(* CoDeSys 2.3 project: cy-wg-016-001.pro *)
(* Title: cy-wg-06 - ClevergyAS *)
(* Author: Andrea Ravasio *)
(* Libraries: Standard.lib 2.12.10 13:48:34, Util.lib 26.9.14 09:12:46, Visual.lib 2.12.10 13:48:34, WagoLibIdent.lib 25.2.13 10:12:16, WagoLibStatus.lib 2.12.10 13:48:32, SysLibFile.lib 2.12.10 13:48:34, SysLibRtc.lib 2.12.10 13:48:32, SysLibSockets.lib 10.2.11 08:20:54, SysLibEvent.lib 2.12.10 13:48:34, SysLibPlcCtrl.lib 2.12.10 13:48:32, SysLibCallback.lib 2.12.10 13:48:32, mod_com.lib 2.12.10 13:48:32, SerComm.lib 31.5.11 07:54:36, Serial_Interface_01.lib 22.4.13 11:50:14, Modb_l05.lib 22.4.13 11:50:12, Ethernet.lib 2.12.10 13:48:32, MBus_03.lib 9.2.13 16:51:58, WagoLibModbus_IP_01.lib 26.5.15 10:20:08, WagoLibMBX_01.lib 20.3.12 15:32:40, LON_01.lib 28.9.12 13:05:10 *)

(* PLC configuration (modules and I/O channels)
VPN_ST2 AT %IX36.0 [BOOLOnX_I] Ch_1 Digital input
LAMP_AL AT %QX22.0 [BOOLOnX_Q] Ch_1 Digital output
KEY_QE_ST AT %IX36.1 [BOOLOnX_I] Ch_2 Digital input
CIR01_EN AT %QX22.1 [BOOLOnX_Q] Ch_2 Digital output
CIR05_AL AT %IX36.2 [BOOLOnX_I] Ch_3 Digital input
AT %QX22.2 [BOOLOnX_Q] Ch_3 Digital output
CIR05_AUTO AT %IX36.3 [BOOLOnX_I] Ch_4 Digital input
AT %QX22.3 [BOOLOnX_Q] Ch_4 Digital output
CIRD02_B_AL AT %IX36.4 [BOOLOnX_I] Ch_5 Digital input
AT %QX22.4 [BOOLOnX_Q] Ch_5 Digital output
CIRD02_B_AUTO AT %IX36.5 [BOOLOnX_I] Ch_6 Digital input
AT %QX22.5 [BOOLOnX_Q] Ch_6 Digital output
CIRD02_A_AL AT %IX36.6 [BOOLOnX_I] Ch_7 Digital input
AT %QX22.6 [BOOLOnX_Q] Ch_7 Digital output
CIRD02_A_AUTO AT %IX36.7 [BOOLOnX_I] Ch_8 Digital input
AT %QX22.7 [BOOLOnX_Q] Ch_8 Digital output
0750-9999/0400-0008 8 DI Generic [Type_1_8_Channels] node 1, in %IB72 out %QB44 {INTTypePAAssignment = PLC; INTTypeModule = plugged}
  CIRD01_B_AL AT %IX36.8 [BOOLOnX_I] I 1: Digital Input
  CIR01_AL AT %IX36.9 [BOOLOnX_I] I 2: Digital Input
  CIRD01_B_AUTO AT %IX36.10 [BOOLOnX_I] I 3: Digital Input
  CIR01_ST AT %IX36.11 [BOOLOnX_I] I 4: Digital Input
  CIRD01_A_AL AT %IX36.12 [BOOLOnX_I] I 5: Digital Input
  CIR01_AUTO AT %IX36.13 [BOOLOnX_I] I 6: Digital Input
  CIRD01_A_AUTO AT %IX36.14 [BOOLOnX_I] I 7: Digital Input
  CIR04_AL AT %IX36.15 [BOOLOnX_I] I 8: Digital Input
  CIR04_AUTO AT %IX37.0 [BOOLOnX_I] I 1: Digital Input
  CIR02_AUTO AT %IX37.1 [BOOLOnX_I] I 2: Digital Input
  CIR03_AL AT %IX37.2 [BOOLOnX_I] I 3: Digital Input
  CTL01_ST AT %IX37.3 [BOOLOnX_I] I 4: Digital Input
  CIR03_AUTO AT %IX37.4 [BOOLOnX_I] I 5: Digital Input
  CTL02_ST AT %IX37.5 [BOOLOnX_I] I 6: Digital Input
  CIR02_AL AT %IX37.6 [BOOLOnX_I] I 7: Digital Input
  AT %IX37.7 [BOOLOnX_I] I 8: Digital Input
0753-0648 LON-FTT [Type_55_1_Channels] node 3, in %IB0 out %QB0 {INTTypePAAssignment = PLC; INTTypeModule = plugged; DataStream = 1F8B0800000000000400ED7D7B6FE2C8D2F7FF8FF47E073F48CFD18C14261808B99C242B0F98095AC0395C921DCD8C90631AF08EB139BE2493FDF46F75B76D6CDCBE10601288A5D52CB1DBD555DDD5BFBA74B97DF9C7AFB9C63D22D3520DFDAAC07F2A1538A42BC658D5A75705C79E14F95AE18FEBFFF73F976D436FE93632; DataStream = 27B282387848B72E7E59EA556166DB8B8BE3E3A7A7A74F4F954F86393D2E974AFCF15F9D765F99A1B95C5475CB96750515FCA7C6E94F15B85BD3989AF2BC058DCF4B17A5D2C529FC7B7251E22F4AB58B52157E14B8BFD449579EA3ABC2BD3C354677AA6DD8A6A1AB4AA50462F4913669188A3347BA2DDB205EDD98E3DF5705; DataStream = 613CE69E0DC7E4147A859B2113D8EB22079E6EAAE6FC4936D19D3F26E7A4A3BEFC886E657B7655A85F7CFFA2DADF95E76289AF159FA6DC8706B290FE8FAC1BDCADACC9FFFC63701D07D85017B28638A1C40B1FBFB7A5EE48474F05AE638C1D0D759DF90332817801C696E3F0E87664F3A7F4F037526C8B5C5BBDEA5E84CB03; DataStream = 345F68B28D5A63605E9DA8C8F4EFC15D3C70ADF175A9C4B1FEBB3C76EF079EE82BC6025DC32DFA2370E74FF48CAFE3FF05AEB6F431FA75CD5F1ED31F3E5FC7098CF94CE309BBEE376F07BA314654B2E583E4A6FF08B369B88964AA5355973566D3D04DFF9196D536949F687C6D9B0E0219BC3F030D3AB23E966DC37CF6DB2C; DataStream = AF049A490BAC56B2763D91358B34F3AFF8AD3A084F349D6E3C94A1BFFD56A286B022D60D07B41196D585AE6A5705DC79813B0E0C08B29F0CF3E79D6CAAF28386ACE0A4ACDC0BDC4AD39897694DB2E6F8DA735E5E559F800AE19B611D4AD523862E75EF0623E3E1EF9189FEEB202B4E9B961AA53FAA3DAF69B4494869824D99; DataStream = DA9449A3D6D0AAEC9A15D52E3E46BB48CB6C1A4689AA7A1FE9E3813A27531BFC33DC4EFE156A17F873B55D0F29487D4481A6C12B2BC2DF9AAA61AAF6F35278FF4AA8651F998FAA8206CFA07982F253379E34349EA2316863E04EE891866A0232C0405EB7F4850393BABC1066190CE04455F0DC5C770D1D98085E0935AD1BFA; DataStream = 449D3A263131B04A16C8B45564AD0E6ACBF2BB5A5196D5EBA1C73E3FDBA8AFFE83AE2B97C7FEEFC0AA3F8E5FF66F16112A498850D9262280E3613B56064030FA6ECB543CF05BBE793828E770901D0E24C7DE2F3CA81D0C1E9C26E1C1E9D6F060A26A08BB0859DC8326B4EDE1A6E9EE81DF748B78E02B7A3A20782433E0C149; DataStream = 8E0787EB1EF0E5C3C1836A121E54B78A07D91D04BCCEB1E9CFE2222CDBBE7950A8E5A070C04E42F9F46050E13C9286A22344A386D25651616164810462FA6F8D2C41C3B2E99B0784D31C100ED74B58376888DC59661C5359BE3C6665AF5F96D24E4E5017F9980C7571CD1435599477AA693BB2C64D1C5DA1AB857BD0605057; DataStream = 33CF6BA59113D66A9E47CE86FF6F2F8F0CCDB3E691A3B43318025F1BB66809D64920C5691969999B02EEADF986BE787946998ED0EB6594A175C68C7284720E0C87050CAFEF23AE890B8793593E4BCA249D6D2D9364836AE1E53B5F64C105AC887D94D1650892CE81E1B08061FF3C86C3C9269D9D2521C3D9B69041D664739E; DataStream = 051404DA300B24B8347334382C34D83B37A17C9EA3C12ED120B38F9003C24102C2FEB907878408491985B3AD651470CC8F32E519B5E73E6D9B05115CB239221C1622EC9F8B703078C097925C0472773B88307B9495D1DC186742859B7A9D1FC12C67CF2704C8E7E87058E8B07FFE029FC3C3EF81871C1BDE3936EC9DE77048; DataStream = D07092080D275BDB85802BA34C3B10041770B3ECDB102EED1C170E0B17F6CF6738A490E2ED02438E0AEF1915F6CE5BC84161D7A0D077168B1C18DE3B30E4EE429E62700769090EE53C0399C3C39EC2C321A519DE343CE4D8F0CEB161EF628A438286B7185394F30C648E0BFBE8331C5248F17681214785F78C0A7BE72DE4A0; DataStream = B06B50C833903930E4EE429E62F00769090E953C0399C3C39EC2C321A519DE343CE4D8F0CEB161EF628A438286B7185354F20C648E0BFBE8331C5248F17681214785F78C0A7BE72DE4A0B06B50C833903930E4EE429E62F007C90587C6CD7D9E80CCD1614FD121CF32ECD06FC0D0202876EE35BC775CC8C3891C16C2B000DE; DataStream = C2ADA1EA79F2F15DE3C2FEF90B3930EC1818F24D891C17727FE1F560E13C0915CEB7060AD6936A2BB32CA0506F36B0B720EA7894321E00E912CF61E1B060217717725C08E1C2971C17725CC8DD857C4FC21BA4B0CF90173EE6E0B0874E43BE27B1C31C0386867C43E2BD8342EE31E498107117F20D89778F0BFBE72CE4C0B0; DataStream = 7B60C8FD85F78E0BB9BF90271E3D50F82CD5F30D891C16727781CB71815BC1857C4322C785DC5DC83724FC410AFB0CF986440E0E7BE834E41B123BCC316068C8130CEF1D14728F21C78488BB906F48BC7B5CD83F67210786DD0343EE2FBC775C38787F2172C75ADE4AE3F9F2B86DE81DD9FC293DFC0DAC91AB2BD7ACEBCBFF; DataStream = FD566F0803E1DBE51FBFE61AF7884C0BA85D15F84FA502877405064C9F5E151C7B52E46B853FAE2FEBB22D6BC6F4FAB2A96A886B59F03F1B99680C8F14B806DCBCF34954310DDC0C4FE15501FF0B7F1BE65CB6FD4635DCA623FF6D9881E70ADCAD6CCFAE0AF58BEF18B54C794EC858DC875F67B58FDF41847B1812EB3BA668; DataStream = 7DEF0F846E43E8353E0DBEDEC29304E6AE0A313858E07A6802FCEA0A4A6C8555BA6FCBF305F0533EE62BC7E5125FE6F8B38B72E9822F17AE57D19AB0C2BCCA7D962D7704FAB05215FB5BED4781234B18C42F70043CAF0AA795028761E9AA4006D644FF759065C3B5479B3E8C710C241447FD416F581F50496168603455853E; DataStream = 49B06E028F8FE0F10287B50CB35FE086BA0A9DFD4BB3FFDDD21F654D1D73966DC2C4423796E1980AFAD7D4FE375BA800FBA2EECC398F3CE66E64E3B9FBA5CE9D3911054086FE2EF29E30BD7839C4EEB0C392C217BDAF4E7557B15C513C49268121E27478CA2A70983B4417833BA427181453641AEA16E905746A0A7361B574; DataStream = 1B4D9149FA6A597D45D664FAC752CE9393CA89271EE98925DCB0DB6F7DE98A8D515BEA7E2970D26462219B108A0AAC5222B8332404C42D87C4755BED5A2217D2391B1680E130272E46B60A7B3209B9914F2E5ECAB9AA69AA8514431F5B99E48499FE5659AE257F0135402BC0CA634DE0E4F11874DC628BD192BA4BF64F58EC; DataStream = 8FB196FB3428C3271EC31E0EF99D645CFFE525CF658F678192E06CFC1800AF6D3E27ADFD44A6313BB6C76DC5E396D543565DEACF0C4C318B32552A011CA85422F2112390A053FD1BA99726202512D1241F1ECE8A0FAACD392EF31C201E759076BB72C203ACAE890CB51721035F8B1375D571206ED44BEC936B5A9C071DD945; DataStream = DD18A3A43595493F2D3D7E29598C7E76A0A57C4049F97DD2D1CFAAED4FCE8A402EF8197359D559EC7F6E0D9A29FA36761F8E67DB9F28DA746DABC49D724404F82760135D814E8302954F3D91BAA00C2F1448278FC68B43F44C2791D63A42542342547D21AA4121026615F09653709374514ED99694D884045988189C31E170; DataStream = 53156533A22F966860CABA25939087380B66BA5C67CC85F26BE43E1E2F1A6900A30793B52E98AF010AE5939330DCAD0302E74CA473C9C44B465B04557003E03EFD115C4A94852FA6E12C3686ECE9221EB2A7A11E3606B034140EABD48BB0F7C1303424EBBB80ADDA5285A0CF17F26F91473380301D7ADAFCDD9B0ECAC75077; DataStream = 2C683B5191367EA1280E2191244A5A249D9B92DC94840078634B32A554365349B6697989C17999CBED02BC63CFF09E804223748389387183C39798112F901C1989E8B33EE6BF44362FC7BDAE54CCBCD00288AD21D5068E43F54770857A19C96A282369D9B2ED247A10490949EF69377E3DDD7E4E92F6104A49F23C3327D98F; DataStream = 95242E25B9E43E3123499BC527246BBB4F42747DE4C61CC5E4BDB2A726A921181993914B2E3E15E11AA45D0BD8471A526C62E1B5E4283D4376D272898D28B1AD656071663221CBF7D26CA43C367DCEB696D57721202691AA98EAC23698063953E0300E90D836E78269CACFDFF8DA0FACEE4D3A43138393F1650ED1ADD2A5C7; DataStream = 8BB75A2CF24800AFFDA758020ABD9EF035453E023D94808B08354F3CCA07B0C6D73865269BE0E02033439298AC8E3A3C90D1F660300DA05CF92C22DCEA9030E6922E99FA8DD05B0A5C66DA5A5FE26FFCC98F953513878E34D925F4EBADD672285E6EB4483FFF71E47146678CAF9E56CF2AB5EA695A6CE60EC37F864223300C; DataStream = 4C6464C4682BD2577D23FD6CAFE541BF1019076969CB302096D7099D33AFD9AD3A22A9A099793B24B07D73BE5DF8A1E8434367AED588411F26F8F80FBD147C68203D52C79E6C51ECA97154FB761BE3C48ABFA963EF4BF82D8235D9B2E9BF29B8A9AD8C8486F4A93DDB3C0470E5F7C8C50F80D8E5F8EA79E9ACC87BE915EF99; DataStream = 379729C50509DB49956E3F8E4BDF7488958AE960AEBBFFB04E84BE01CCF2812D3E7E59837256098648887B04E738D9F78B09F9702084189B95D885561FD5B1236B1C5EB0649D6E21674CD9C5144BF1A9A328AFF040693B3983F8C4640ABFFC9AFCF2BBE1B79C95DFF29AFC9677C36F252BBF9535F9ADEC86DF6A567EAB6BF2; DataStream = 5BDD0DBF2759F93D5993DF93DDF05BCBCA6F6D4D7E6BBBE1F7342BBFA76BF27BBA457EB37178969EAC67BA36F0ECD92B83EFF9CB593F7F651CE6130C5D1AEFFC8E8C5E6650E613AC5E2AF33BB28099119A4F3081A9CCEFC81C66866B3EC11EA632BF23DB9819BBF904E398CAFC8E0C656620E7132C652AF399ADE6D6AAFEBC; DataStream = 88C0CFC2E08278BCC13167EE65A6C40378D375E43E4CB9F737809E916C1E717343B76747DC587E3EE2668683AFA8BA63A3238E160467CC9A66CF9C554AB8CA9FB139F415C9EC882798438B8AF94C1E4B4A07968312AF930E5C2B7EF5C4E8E0015D277E6506E5734A255EF748831D09535926CA646631749C28CC487C2C2756; DataStream = 3CC0ED1D8951F683EA1B50EC75E4A8B2E4981122F182E0FB3B92E4E4DCD72EB23837AE919DBB6412F48BB4D8B93C7D0A326BC8C32C1C72B12A29871578BD6193FC4D204FCE2F77ECCFFCAD1F01849DBF7CCB1E8FD5DC07AE9D64CCDB865BFFB146C2DC7B26215F1E1548F31F7ADD1C799CC01BAE214FBCF512E458E08DF3E3; DataStream = 2FDCA7A2AF1EC66C7BACF376844108D1ED8FD80D2BDA28F3DE3DA92721EA3FC25B61A172924A39E43154C28BCD8ED97EA3352589756BCBFE92365165BF9BF80A93D3AC222EDC42A591861E9196A56AC62F6D224FA44BCA2C630B779B24ED22D45DBCC467BFE9253F0C14DDBB75EA69981B5A440F47B631C2389BA4B7EAB253; DataStream = 4E911D0B83AD0BCBA9F2529CAD129CBDC329F61890ADB240F68EEE9DA5EE48B2B771DC9DB7951D701F6AABBF056A9932AFB195C3045A221929934908C57E2FACD22026396E89D34E26A232A2983D085D7826A8EE67ECC23361730F831776F1D09E462FEC12A03D0E5FCAEC3DF8B5E2976DA3D9F9796086FC57C1D7A9686206; DataStream = FEF320ADADBD7D1E34B1D4FFD3D43978D86B18DAC06319CC2DBB5C8B7A8E2E8DD735BA09A3B0865E26F8C784F466067883903B5CCEEB3A9FE7BEF925B5960BC352E3E2D32C45F2F07C244A5DE0D3CF9079E4D5F3ECBE38B287E4F1F13DF8DE5820D2796AA924E315A3A7D1C24EC988FA9A4AAAABF1D42DDF53DCFD3117BE90; DataStream = 196AB5C238C3CCCB81C0B1555A3EC82CDFAB5AD6846E5D277D47CA0DB45F7E940CC4CEA3C0692CA1E3245A8D239FF21B4A18FCC62C814B9875164EB9CA0CA1D327241C42338D74B8DBA410DA0875171F42E3487543450C6C1E9597BB47E79515C95F9C90C49A187E85A8165444F7C59B89264FB39BB983D1C6D4620D37675B; DataStream = 6C35C810A56F4432154FA554D8BC6F612B95CF2684A7CE5B9064B9867E7F294743B53091F126728C5D1AAF52CE213976D198148957666D2285E1D8F805334AE8558A3BA405D28B8A6A2A8EBA915E194067E4D27995420F774E2C7A72E21626C5A5F42A851F1DA4CC645D858E8B13D9D1369A99B94F6B4468BD4A314813A1F1; DataStream = 83ACFC047154CD31379A9F894B6BE4D2FA4D657FD223328BA6AC4FB332CF0CC90DA03222545EC5920CC1AE6E410A0793D9A518291644C4EFAE9A6BAF0FA62CC8A7B5CBF591625186E49B4145DB28CE916C655F2031B38389E19D1697D8AB5896BA319F3BBA7BD481B5E6C267CAA500C51D2CFAEC36A6097DA331D8186D52B4; DataStream = B33B624C61B01C234C6964EFCC0F4B2B2FF4E428AA7A718139C4870F6D20932FCE48D5471EC157B137F424E22298F24DE4D1089511FBF0CE5DD8988EAC3B80698AA1DBA6A165649D999399134A2397D22B452D0BF0C9E8D6FD0692802A793539BFDFD05019B0D136D57156F08A13C323F32A16A68716866917E7B2F5731331; DataStream = 4C426684C9BC8A55F13852F569117F1D6B1359164B5AE44B5BAF62538202619BB02D8130AD57B12A6433A4A81BB63A792E8ED70BF59952D12D104A70B4DBB83FC5AAF490C57EDF37D3C2817B80C7F3858692774E5F7044DF1917342D7E2924EED37C44E30CAF6D30B7D802CFEFE2F4AD0D12FDCB77B0C907345F9056B5DC07; DataStream = 57F28FA4D4856655D14E760D97652BB1D546AB3B84F1A546EEA478EF487CA619F79509FA3F722492A3695EF95AAA5EF5373953387CD854D25923ABF51F71C74FA51C36E20B4ADA92F3ED363C5FC54D8F7B5B0427190B5FCAA7B5D07934E5D30AEF6F2DE22FB6E0BD0712BBACFD8E45E0532EE1C1F0A6BD9CF4DAC51881278E; DataStream = 2CAE8E344B75B26C31925D1EF2094A3B301067214566CEF9CD9D50E7E6310708C49D3116FEE065D214FBE413B674AAB1B36F5D5F06DA87FFE2965F4E18C853F7AC9FE506D7F525ADAC0B25E439770947256AF646DD61BBC0F5E427D2860ED171984A1F53D76D55D638595170EC6522BC77CD2427DD8ADDD1401AF5C56E2303; DataStream = A527BCBF9B42AA27D6C5D69D18E432CA645D332CC4C93A80BBFC88DCA3C79864EB6DA92F8E9AAD7688623981E218615B984EB321B6C54194742542BA478EEC0436C7E4933486F9EC7D4F8049BDD182211848BDAFB0EEA43F87B741E2D5287160D998AF3955A39E10A47A9242758D695BA14C0FD83B0E683453BD6B41F5F6CF; DataStream = 0D5C57BBFB19B49B9485D8F878D3093239CB210282198A21F857530411FF8C9069F833A919C64F7CE46F1A253A97845692628BA669981C3E85738174ECB5C4AA619F0E7D5368B59335DB27395E613A9953B1D74B56EBF050AA3AB7CCADC48FE5B0DB107BF7B88E2A49A97D96B13EC3281C630D4C198D96B4CA7254ADC32CE3; DataStream = 9720C71CC9A330290E5A1D511A0E56C9D62264EF55582D4F9C45F04E411CC2ECC710BD6F751BD2FD2ACDD308CD954359FD042393A8301CDCAC923C8B92A4AB991A2AC3069D5DE0B019B11103A8D6EB62BF0F5326DCAD28D9790A603CA0670390549498A72200E9BE28FE396A75EF8436DEB60F2C885274CEDCD6F7428BE975; DataStream = 86EF0748F1D9B0E7D4C59ED03B266116868B31F6E1FCF99D815622E6040BEDD18D28808A876128BA7856494E0CC38E25D994A4C12AC9E83A6FA007674A8E17C41FF4C2127EC0B32CEBF435858F31C41BE2E7E19730ED282CB502541DCA7A26E2AD6E530AD38E4E70FFD9021F727DC6FB5FFB03B113ED22BA3E0733F76C694E; DataStream = B538B7D620862868E450646966318A2621B232B8F83A982EDD3D44299B0C75A98BBF961652DC62140F714F6344B690A12B6332D1549D890540526A36DBAD6EC8252946F58F1687E2E25A954EAA8EBFF407233F979F61F9726368691B44AAC0868907431CA0F34C36C74F32DE3BA1D7E2441C76FFEC4AF7DD103F51E5F5AC7B; DataStream = E09D2A7718E5154E09722D90823F61398EEB34DD11E81ADC2AE505CE2CE84C6B80494A78B61AAD013916767539EB3E4B6B9215DA9D20DD24DF6060D8B276ECD5129042D047EC5B93FE78EE034EE3183A74452ACCC0D85B9CD718E60B9F4167235D06B4891BB5813418F5EFEA84273ED9A948E485B941BE42BF9CEC5C24D267; DataStream = 6E8BACD0AF247B186E7134586DB7409A4E9A8664936386FC40BE0D76BBDD1980FBDF0B0F4F141A92C8C78D4E907C39D9E1A0E467EA74B606FB37AD2F376CFE19DE4752077102843A28A7F822CC014A1BF98862461D1136E1B4318F6824C34EC58C49EA70479866D8D718DAA9231DE53BBA549B8004ABA014E768B47A986488; DataStream = 20CBF10782806AC5EC446F7B628470745162C24513E16F0D8FC14D379C0770D73F90FA878F99BA19F43E87709F678500813EC003C6086319E4FB1D1E607F409FA69F8EC0C898AAFE5383400123B89560E270D7FDE1ED5DA8EBE8AA0D8B8777B8892B9E7D1407627F1019C6E8E28DE967BD19237DB1A62DBA9643FDCD692A8E; DataStream = 43FAA36A1A3A7EDF04701B9B26A45BD489A02F104368A7CCD8B187CB82D8BDAB4B9DDB5147F82BC44174D18738901F74EC486A6035168E9D49D88ED46D0DA41E31C421BBC70847C2C2FA3615A6119971469EF421B4BA78F6C45EC8DB2B337214F88BBE9CBC58689EDB151B5062DAC200FE85E04F0AC7EB51D62588284D4A2B; DataStream = 7554A2F4A27C527AE0039244451AC57BA1D76D75439146A59C2D443B7343B4C83BF26B66886EB3E43FDBC6132EA2A12B65B1F28E3D93665BBC13DBA3E878FBB79826227837C9EBF3DB318D41F06E92BF7603A6E545625592FDB4B63A415C5F9E202046EC02B16416F7E1B350C78703FB87149499E079BBE289446DC22DFD8E; DataStream = F673A64E2A719D9493DD3542B41F3006D41E47E857E3E85792FD35427F400DDA7193D4067E68A8D642939F3F467B3989EBA59AECB4915E6E019E08F7471CD996A8E3CC990278224248B0C0701C275C2DAEDB5AB22B47BA899B91B338A267C96E5C1CEFBD41F788EA00FC4A1A44BE14AB70A514478FF44DC86B140BBCE5C2EA; DataStream = 2676D4F81AC3E74B853ACC0EC1BAC8CB4C6B625DEF3F19B04E243599EE8B5364F3C34473E311AEF845416CCA52AF23B41959712B402FE6D946AB2F7C6E8B8D64D4A385411E67DE9B464C82C3DB8630C03BEBC260D84F46C15B64E224934FD62B358CA1DC17DB4DE2082563A09BCB9343473C25B12AB4855E2719F65CF9DDF7; DataStream = A8F05141B4B88949B627DE4ABD017818FD3F93714EF24AC6126748BA03EBDF6A88C99816D29D184A62174F75326AF55C8DA35392A278BDCE1D93BD282AD549A89A457FEA6D51E831D4270A4A219A6EF95F02C9C83433B0C61D45AA3BA49A48F54EC76252263461FD0D5ACDAFEEF0361838C35A952FEB83B95C199B4C212499; DataStream = 907C13AEF5E4FC5A4F66571DA13BC469D0412F1CB7451759B4030C55A4B222A9839ED89160C5453A60EC39D10E02D56AB84285A4F5A8181375EAB860BDA04E09F90E23B3DBDB9EF4A52784273FBA1CA93E911AACA25783456AD2B80FE1C22CA68DF1F5AC27F6C5F0D60763B5FE428A03D46967FEB6034898B880A3A4A30B98; DataStream = 4A011028739A314DE4B42D85FC7F462CD93664885967FE3C2C53BD7887B15FBF1DE01BF49B63315DB525A1C19C00C6AE95A393CE14C734C1BBD0F0CEA83C86BEDCDE3F71AD49889B27D9E266B246633FACDFDAF31134502DEE49D5704C6B8145E74C47A77BB7A631A78FE3D7F671EA7EF9FCA7B8111F7659CC3322D11BA093; DataStream = C2FDC0E76CE156CD85C796942661B32FE3EFBC53AD001F0B4605A7FDF18DA058C14789684F10FF210E6C53BA5837427BC0948B65FA812F3359B4E5D03EA0A94A463B7640C17E0B3D76E7511C1BEA9AA781717DC7D9F66E9CE29519684697A3453AD2D12F1B2F1DE2EA1A0BCF23FC803779DCA23FECFB1EC10AB048F921DC3D; DataStream = A20F700FF86D80230ED9CAA78F7835A7E9C3EAE4CF1DF06F1F10F7AFFF3A86FD6F75AC21FA0BEF18D05F745EDDAB784B4851D0C2A64AEF6AC91167E054C0936A516DC03A0334D5A96E98A012A16E4D643BA66E614A0CFAAE464E6C9CA8206344BE483A097517E7AD0DC45BE6F05733BADE55D7F5762BCCD80EF7639CC38DA3; DataStream = 860C2E779D9A2B9C56941DDB2004308CE0CFB0E95384F7CEED2784F450FE07E7EF98A686742A0C0752141D904C2A260C5D63161A91276F446190EC870B4B2E8A2E142BC00E4DF93CE19A6A761D0921DFE975BF8CEE7B9D700D13A3F6CA30B4545EEB92D44EF6C399BCEAEA7406119C634E1366ADF5E5060062D8FB22267BE5; DataStream = CC1E705E5531D81E08218FB3A8ABDC339C81A562E02D4ED7ADA1E3E2D80BC78E5700A9D94CF1D5FDF8F901618238E661A75E09BDD590276AF345583C53F0209E712D844D4B4A3E909F0B67BE60BA2B84B2D8117B5F226AC7D81E52FD51A0494504203391C15A0378E0A21DA6EF4ABA680ADD91D46D7F4D71E55D957B52ED19; DataStream = C94EE314BF413B75CD777C0F3D313AA10CDFBEA5A0E25CFE89BBA115A431F45A7531C58577EB5BC960A792EB087F451736C36387B135E6A0BF18298EF178249315EB5257EA7C4D71D31B68E6CCD5B11F6224D36C8837C3CE4A055074D5D501781FCC0CE4EA42BBF5B90711768ADFBDD45E255D6CA2B191D966AC319F28AC2D; DataStream = 307419A882C512D23673FC29A52C24CC79844776AA6E747357273E72BC55F01B243ACF143AA5645AFEFD882B1BB6C7C7E112E8635CA9777D49EAF55A16FC0F1C02B7F6BA0181C61D322D6888B5E51350C3CD6851777301514193D411F96D4E70938EFCB761061E0386657B06BA75F1DDE59C50B1B80FBFCE6A1FBFB70DFDDE; DataStream = 307F5ADF4981F6775CA3D3107A8D4FCD5BB706AD05CC944A1CEB3F90154D805D88AF125BE10F38F4F12718F0F23CE62BC7E5125FE6F8B38B72E902D62B48EFE8C4D79335E8917CEE9971CDF75EBC5A77FC9D3C4EF2833A5557D485ACC59C5AD00781F027EFDCF691027C18FC0E785C32AE1AA5EF15207C6016FDA875A0D3D5; DataStream = 8394A23DE98F6ACFBB8B0735703856B4EE3FA5DBD503B5E2D33BFAA3E17D5C3CD86985D969B813FF651EA284C992E126205DA893D32C9DD4429D24CA815B6059C29D543374721AEA6479265EAC28B7C6CA78B92B36A27CAC6BCBD57B5CC71B99C6F4FAC70FF8A38DDF8580653C911574FDFF0124FCD43EE1460100; DataStream = .; DataStream = .; DataStream = .; DataStream = .; DataStream = .; DataStream = .; DataStream = .; DataStream = .; DataStream = .; DataStream = .; DataStream = .; DataStream = .; DataStream = .; DataStream = .; DataStream = .; DataStream = .; DataStream = .; DataStream = .; DataStream = .; DataStream = .; DataStream = .; DataStream = .; DataStream = .; DataStream = .; DataStream = .; DataStream = .; DataStream = .; DataStream = .; DataStream = .; DataStream = .; DataStream = .; DataStream = .; DataStream = .; DataStream = .; DataStream = .; DataStream = .; DataStream = .; DataStream = .; DataStream = .; DataStream = .; DataStream = .; DataStream = .; DataStream = .; DataStream = .; DataStream = .; DataStream = .; DataStream = .; DataStream = .; DataStream = .; DataStream = .; DataStream = .; DataStream = .; DataStream = .; DataStream = .; DataStream = .; DataStream = .; DataStream = .; DataStream = .; DataStream = .; DataStream = .; DataStream = .; DataStream = .; DataStream = .; DataStream = .; DataStream = .; DataStream = .; DataStream = .; DataStream = .; DataStream = .; DataStream = .; DataStream = .; DataStream = .; DataStream = .; DataStream = .; DataStream = .; DataStream = .; DataStream = .; DataStream = .; DataStream = .; DataStream = .; DataStream = .; DataStream = .; DataStream = .; DataStream = .; DataStream = .; DataStream = .; DataStream = .; DataStream = .; DataStream = .; DataStream = .; DataStream = .; DataStream = .; DataStream = .; DataStream = .; DataStream = .; DataStream = .; DataStream = .; DataStream = .; DataStream = .; DataStream = .; DataStream = .; DataStream = .; DataStream = .; DataStream = .; DataStream = .; DataStream = .; DataStream = .; DataStream = .; DataStream = .; DataStream = .; DataStream = .; DataStream = .; DataStream = .; DataStream = .; DataStream = .; DataStream = .; DataStream = .; DataStream = .; DataStream = .; DataStream = .; DataStream = .; DataStream = .; DataStream = .; DataStream = .; DataStream = .; DataStream = .; DataStream = .; DataStream = .; DataStream = .; DataStream = .; DataStream = .; DataStream = .; DataStream = .; DataStream = .; DataStream = .; DataStream = .; DataStream = .; DataStream = .}
  AT %IB0 [BYTEOnB_I] First Byte of 24
  AT %QB0 [BYTEOnB_Q] First Byte of 24
0750-0464#04 2/4 AI RTD / ADJ./ HA [Type_44_4_Channels] node 4, in %IB68 out %QB44 {INTTypePAAssignment = PLC; INTTypeModule = plugged}
  S01 AT %IW12 [INTOnW_I] Channel 1
  S02 AT %IW13 [INTOnW_I] Channel 2
  S03 AT %IW14 [INTOnW_I] Channel 3
  S04 AT %IW15 [INTOnW_I] Channel 4
0750-0464#04 2/4 AI RTD / ADJ./ HA [Type_44_4_Channels] node 5, in %IB92 out %QB68 {INTTypePAAssignment = PLC; INTTypeModule = plugged}
  S05 AT %IW16 [INTOnW_I] Channel 1
  S08 AT %IW17 [INTOnW_I] Channel 2
  S06 AT %IW18 [INTOnW_I] Channel 3
  S07 AT %IW19 [INTOnW_I] Channel 4
0750-0464#04 2/4 AI RTD / ADJ./ HA [Type_44_4_Channels] node 6, in %IB100 out %QB68 {INTTypePAAssignment = PLC; INTTypeModule = plugged}
  S09 AT %IW20 [INTOnW_I] Channel 1
  AT %IW21 [INTOnW_I] Channel 2
  AT %IW22 [INTOnW_I] Channel 3
  AT %IW23 [INTOnW_I] Channel 4
0750-0478 2 AI 0-10V 16 Bit S.E. [Type_8_2_Channels] node 7, in %IB108 out %QB68 {INTTypePAAssignment = PLC; INTTypeModule = plugged}
  VRD01_ST AT %IW24 [WORDOnW_I] I 1: Analog Input
  VRD03_ST AT %IW25 [WORDOnW_I] I 2: Analog Input
0750-0478 2 AI 0-10V 16 Bit S.E. [Type_8_2_Channels] node 8, in %IB116 out %QB68 {INTTypePAAssignment = PLC; INTTypeModule = plugged}
  VRD04_ST AT %IW26 [WORDOnW_I] I 1: Analog Input
  AT %IW27 [WORDOnW_I] I 2: Analog Input
0750-0556 2 AO ±10V [Type_14_2_Channels] node 9, in %IB120 out %QB68 {INTTypePAAssignment = PLC; INTTypeModule = plugged}
  VRD01_CTRL AT %QW12 [WORDOnW_Q] O 1: Analog Output
  VRD03_CTRL AT %QW13 [WORDOnW_Q] O 2: Analog Output
0750-0556 2 AO ±10V [Type_14_2_Channels] node 10, in %IB124 out %QB68 {INTTypePAAssignment = PLC; INTTypeModule = plugged}
  VRD04_CTRL AT %QW14 [WORDOnW_Q] O 1: Analog Output
  AT %QW15 [WORDOnW_Q] O 2: Analog Output
0750-0650/0003-0000#03 RS 232 C Interface (Adjustable), 3 Byte [Type_21_1_Channels] node 11, in %IB124 out %QB72 {INTTypePAAssignment = PLC; INTTypeModule = plugged}
  AT %IX28.0 [BOOLOnX_I] Transmission acknowledgement
  AT %IX28.1 [BOOLOnX_I] Reception request
  AT %IX28.2 [BOOLOnX_I] Initialization acknowledgement
  AT %IX28.3 [BOOLOnX_I] Input buffer is full
  AT %IX28.4 [BOOLOnX_I] Number of received characters Bit 0
  AT %IX28.5 [BOOLOnX_I] Number of received characters Bit 1
  AT %IX28.6 [BOOLOnX_I] Number of received characters Bit 2
  AT %IB57 [BYTEOnB_I] Input data Byte 0
  AT %IB58 [BYTEOnB_I] Input data Byte 1
  AT %IB59 [BYTEOnB_I] Input data Byte 2
  AT %QX16.0 [BOOLOnX_Q] Transmission request
  AT %QX16.1 [BOOLOnX_Q] Reception acknowledgement
  AT %QX16.2 [BOOLOnX_Q] Initialization request
  AT %QX16.4 [BOOLOnX_Q] Number of characters Bit 0
  AT %QX16.5 [BOOLOnX_Q] Number of characters Bit 1
  AT %QX16.6 [BOOLOnX_Q] Number of characters Bit 2
  AT %QB33 [BYTEOnB_Q] Output data Byte 0
  AT %QB34 [BYTEOnB_Q] Output data Byte 1
  AT %QB35 [BYTEOnB_Q] Output data Byte 2
  AT %IX30.0 [BOOLOnX_I] Transmission acknowledgement
  AT %IX30.1 [BOOLOnX_I] Reception request
  AT %IX30.2 [BOOLOnX_I] Initialization acknowledgement
  AT %IX30.3 [BOOLOnX_I] Input buffer is full
  AT %IX30.4 [BOOLOnX_I] Number of received characters Bit 0
  AT %IX30.5 [BOOLOnX_I] Number of received characters Bit 1
  AT %IX30.6 [BOOLOnX_I] Number of received characters Bit 2
  AT %IB61 [BYTEOnB_I] Input data Byte 0
  AT %IB62 [BYTEOnB_I] Input data Byte 1
  AT %IB63 [BYTEOnB_I] Input data Byte 2
  AT %QX18.0 [BOOLOnX_Q] Transmission request
  AT %QX18.1 [BOOLOnX_Q] Reception acknowledgement
  AT %QX18.2 [BOOLOnX_Q] Initialization request
  AT %QX18.4 [BOOLOnX_Q] Number of characters Bit 0
  AT %QX18.5 [BOOLOnX_Q] Number of characters Bit 1
  AT %QX18.6 [BOOLOnX_Q] Number of characters Bit 2
  AT %QB37 [BYTEOnB_Q] Output data Byte 0
  AT %QB38 [BYTEOnB_Q] Output data Byte 1
  AT %QB39 [BYTEOnB_Q] Output data Byte 2
0750-0653/0003-0000#03 RS485 Interface (Adjustable), 3 Bytes [Type_21_1_Channels] node 13, in %IB128 out %QB80 {INTTypePAAssignment = PLC; INTTypeModule = plugged}
  AT %IX32.0 [BOOLOnX_I] Transmission acknowledgement
  AT %IX32.1 [BOOLOnX_I] Reception request
  AT %IX32.2 [BOOLOnX_I] Initialization acknowledgement
  AT %IX32.3 [BOOLOnX_I] Input buffer is full
  AT %IX32.4 [BOOLOnX_I] Number of received characters Bit 0
  AT %IX32.5 [BOOLOnX_I] Number of received characters Bit 1
  AT %IX32.6 [BOOLOnX_I] Number of received characters Bit 2
  AT %IB65 [BYTEOnB_I] Input data Byte 0
  AT %IB66 [BYTEOnB_I] Input data Byte 1
  AT %IB67 [BYTEOnB_I] Input data Byte 2
  AT %QX20.0 [BOOLOnX_Q] Transmission request
  AT %QX20.1 [BOOLOnX_Q] Reception acknowledgement
  AT %QX20.2 [BOOLOnX_Q] Initialization request
  AT %QX20.4 [BOOLOnX_Q] Number of characters Bit 0
  AT %QX20.5 [BOOLOnX_Q] Number of characters Bit 1
  AT %QX20.6 [BOOLOnX_Q] Number of characters Bit 2
  AT %QB41 [BYTEOnB_Q] Output data Byte 0
  AT %QB42 [BYTEOnB_Q] Output data Byte 1
  AT %QB43 [BYTEOnB_Q] Output data Byte 2
0750-0461/0000-0007 2 AI PT100 Resistor Measur. 10R-5k0 [Type_8_2_Channels] node 14, in %IB132 out %QB84 {INTTypePAAssignment = PLC; INTTypeModule = plugged}
  VRD02_ST AT %IW34 [WORDOnW_I] I 1: Analog Input
  AT %IW35 [WORDOnW_I] I 2: Analog Input
0750-9999/0500-0002 2 DO Generic [Type_10_2_Channels] node 15, in %IB74 out %QB45 {INTTypePAAssignment = PLC; INTTypeModule = plugged}
  CIR05_EN AT %QX22.8 [BOOLOnX_Q] O 1: Digital Output
  CIRD02_B_EN AT %QX22.9 [BOOLOnX_Q] O 2: Digital Output
0750-9999/0500-0002 2 DO Generic [Type_10_2_Channels] node 16, in %IB75 out %QB45 {INTTypePAAssignment = PLC; INTTypeModule = plugged}
  CIRD02_A_EN AT %QX22.10 [BOOLOnX_Q] O 1: Digital Output
  CIRD01_B_EN AT %QX22.11 [BOOLOnX_Q] O 2: Digital Output
0750-9999/0500-0002 2 DO Generic [Type_10_2_Channels] node 17, in %IB75 out %QX22.10 {INTTypePAAssignment = PLC; INTTypeModule = plugged}
  VRD02_OP AT %QX22.12 [BOOLOnX_Q] O 1: Digital Output
  VRD02_CL AT %QX22.13 [BOOLOnX_Q] O 2: Digital Output
0750-9999/0500-0002 2 DO Generic [Type_10_2_Channels] node 18, in %IB75 out %QX22.12 {INTTypePAAssignment = PLC; INTTypeModule = plugged}
  CIRD01_A_EN AT %QX22.14 [BOOLOnX_Q] O 1: Digital Output
  AT %QX22.15 [BOOLOnX_Q] O 2: Digital Output
Fieldbus variables [FB_VARS] node 1, in %IB0 out %QB0
Flag variables [FLAG_VARS] node 2, in %IB0 out %QB0
Modbus-Master [MB_MASTER] node 3, in %IB0 out %QB0
*)

(* Global variable list: Global_Constants *)
VAR_GLOBAL CONSTANT

	Plant_NAME			: STRING :='cySN:16 cyVER:1 - ';
	Plant_SN			: DWORD  :=16;	(* S/N Impianto di telecontrollo *)
	Plant_SW_VER		: WORD   :=1;		(* Versione SW installata *)


	(* Colour defines *)
	COLOR_RED			: DWORD	:= 16#2020F0;
	COLOR_YELLOW		: DWORD	:= 16#20F0F0;
	COLOR_GREEN			: DWORD	:= 16#20F020;
	COLOR_LIGHT_GREEN	: DWORD := 16#006000;

	(* Parameters *)
	Plant_DefaultTAmb	: INT	:=100;		(* [.1°C] Temperatura ambiente di default in caso di rottura sonda *)
	Plant_MaxRunTAmb	: INT   :=210; 		(* [.1°C] Temperatura ambiente massima funzionamento impianto *)
	Plant_AntiFreezeTAmb: INT   :=-40;		(* [.1°C] Antifreeze temperature, start circulators *)
	Plant_VRD_TAlarm	: INT   :=850; 		(* [.1°C] Temperatura di allarme VRD, blocco *)
	Plant_VRD_TMax		: INT   :=800; 		(* [.1°C] Setpoint massimo per uscita VRD *)
	Plant_VRD_TDefault	: INT	:=300;		(* [.1°C] Temperatura di default in caso di errore climatica *)
	Plant_CirOffDelay	: TIME	:=T#30m;	(* (Def.T#15m) Ritardo spegnimento pompe per ricircolo caldaia *)
	Plant_CirOnDelay	: TIME	:=T#15m;
	Plant_MaxWaterLoss	: WORD  :=2;		(* [lt/h] Massima perdita del circuito *)

	(* Filesystem *)
	FilesPath  			: STRING :='S:\';

	(* TCP Logger *)
	Logger_SERVER		: STRING:='';
	Logger_IP			: STRING:='192.168.100.3';
	Logger_PORT			: WORD  :=80;
	Logger_GETSTART		: STRING:='GET /cygmsrv/hsgm.ashx?';
	Logger_GETEND		: STRING:='$R$N$R$N';
	Logger_CHECK		: STRING:='True';
	Logger_CRLF			: STRING:='$R$N';
	Logger_DataFile		: STRING:='S:\LOG.DAT';
	Logger_DataFileOld	: STRING:='S:\LOG.BCK';
	Logger_IndexFile	: STRING:='S:\LOG.IDX';
	Logger_ConnRetries	: BYTE:=5;
	Logger_RecoverMsgs	: BYTE:=25;

	(* TCP Remote *)
	Remote_PORT			: WORD  :=10;
	Remote_WELCOME		: STRING:='Connected$R$N';
	Remote_OK			: STRING:='OK$R$N';
	Remote_ERROR		: STRING:='ERROR$R$N';

	(* TCP Sockets *)
	MAX_SEND_TCP_SERVER					 : DWORD:=3000;(*60000*)
	MAX_RECEIVE_TCP_SERVER				 : DWORD:=3000;
	MAX_RECEIVE_TCP_SERVER_SOCKET	 	 : DWORD:=1500;
	MAX_SEND_TCP_CLIENT					 : DWORD:=3000;(*15000*)
	MAX_RECEIVE_TCP_CLIENT				 : DWORD:=1500;
	MAX_RECEIVE_TCP_CLIENT_SOCKET		 : DWORD:=1500;
	MAX_RECEIVE_UDP_SERVER				 : INT  :=1472;
	MAX_RECEIVE_UDP_CLIENT				 : INT  :=1472;
	CONNECT_WATCHDOG_TIME				 : TIME :=t#10s;

END_VAR

(* Global variable list: Global_Retain *)
VAR_GLOBAL RETAIN PERSISTENT
	Mode_Manual : BOOL := FALSE;

	GRU01_Clima	: typ_Clima;

	VRD01_Clima : typ_Clima;
	VRD02_Clima : typ_Clima;
	VRD03_Clima : typ_Clima;
	VRD04_Clima : typ_Clima;

	Ctl01_Counter	:	DWORD;
	Ctl02_Counter	:	DWORD;

END_VAR

(* Global variable list: Global_Variables *)
VAR_GLOBAL

	SYS    : typ_SYS;
	Logger : typ_Logger;

	Lamp	:	PLANT_STATUS;
	T_AMB	:	INT;		(* Environment temperature *)

	(**** PLANT OBJECTS ****)
	(*...*)
	GRU01	:	obj_CAL_VT300GW2 := (ID:=1);

	(* Frigo *)
	FRG01	:	obj_MODBUS_FRG_AER485 := (ID:=1, Address:=1);

	(* Water counter - 2 PULSES/LITER *)
	CTL01	:	obj_CTL	:= (ID:=1, Peso:=5);
	CTL02	:	obj_CTL	:= (ID:=2, Peso:=5);

	(* Heat counter *)
	CTB01	:	obj_MBUS_CTB_SHARKY775 := (ID:=1, Address:=16#53090390);

	(* Cronothermostat *)
	THER01	:	obj_CRONTER := (ID:=1, Local_MaxRunTAmb:=250,Histeresys:=10);
	THER02	:	obj_CRONTER := (ID:=2, Local_MaxRunTAmb:=250,Histeresys:=10);
	THER03	:	obj_CRONTER := (ID:=3, Local_MaxRunTAmb:=250,Histeresys:=10);
	THER04	:	obj_CRONTER := (ID:=4, Local_MaxRunTAmb:=250,Histeresys:=10);
	THER05	:	obj_CRONTER := (ID:=5, Local_MaxRunTAmb:=250,Histeresys:=10);
	THER06	:	obj_CRONTER := (ID:=6, Local_MaxRunTAmb:=250,Histeresys:=10);

	(* Crono *)
	CRON01	:	obj_CRON := (ID:=7);

	CronEd	: 	obj_CRON_EDITOR;

	(* Pump *)
	CIR01	:	obj_CIR	:= (ID:=1, OnDelay:=T#1m, OffDelay:=T#30m);
	CIR05	:	obj_CIR	:= (ID:=2, OnDelay:=T#1m, OffDelay:=T#30m, ExtStatus:=FALSE);

	(* Double pumps *)
	CIRD01	:	obj_CIR_DOPPIO_new := (ID:=1, OnDelay:=T#1m, ExtStatus:=FALSE, Mode:=1);
	CIRD02	:	obj_CIR_DOPPIO_new := (ID:=2, OnDelay:=T#1m, ExtStatus:=FALSE, Mode:=1);

	(* ModBus Pumps *)
	CIR02	:	obj_MODBUS_CIR := (ID:=1, Address:=1, OnDelay:=T#1m, OffDelay:=T#30m);
	CIR03	:	obj_MODBUS_CIR := (ID:=2, Address:=2, OnDelay:=T#1m, OffDelay:=T#30m);
	CIR04	:	obj_MODBUS_CIR := (ID:=3, Address:=3, OnDelay:=T#1m, OffDelay:=T#30m);

	(* Valves *)
	VRD02	:	obj_VRD_POT_new	:= (ID:=2, fFeedback:=FALSE, Local_VRD_TAlarm:=800);
	VRD01	:	obj_VRD_new 	:= (ID:=1, fFeedback:=TRUE, Local_VRD_TAlarm:=800);(*,Ctrl_ErrGate:=200,ReducedRange := TRUE ); (* ReducedRange := TRUE);*)*)
	VRD03	:	obj_VRD_new 	:= (ID:=3, fFeedback:=TRUE, Local_VRD_TAlarm:=800); (*,Ctrl_ErrGate:=200,ReducedRange := TRUE ); (* ReducedRange := TRUE);*)*)
	VRD04	:	obj_VRD_new 	:= (ID:=4, fFeedback:=TRUE, Local_VRD_TAlarm:=800);(*,Ctrl_ErrGate:=200,ReducedRange := TRUE ); (* ReducedRange := TRUE);*)*)





	(* Temperature probes *)
	TPV01	:	obj_TPV := (ID:=1);
	TPV02	:	obj_TPV := (ID:=2, IN_WMIN:=50 ,IN_WMAX:=800);
	TPV03	:	obj_TPV := (ID:=3, IN_WMIN:=50 ,IN_WMAX:=800);
	TPV04	:	obj_TPV := (ID:=4);
	TPV05	:	obj_TPV := (ID:=5);
	TPV06	:	obj_TPV := (ID:=6);
	TPV07	:	obj_TPV := (ID:=7);
	TPV08	:	obj_TPV := (ID:=8);
	TPV09	:	obj_TPV := (ID:=9);

	(* Zigbee temperature probes *)



	ZTHL01	:	obj_ZTHL := (ID:=1, Address:=11);
	ZTHL02	:	obj_ZTHL := (ID:=2, Address:=12);
	ZTHL03	:	obj_ZTHL := (ID:=3, Address:=13);
	ZTHL04	:	obj_ZTHL := (ID:=4, Address:=14);
(*	ZTHL05	:	obj_ZTHL := (ID:=5, Address:=15); *)
	ZTHL06	:	obj_ZTHL := (ID:=6, Address:=16);
	ZTHL07	:	obj_ZTHL := (ID:=1, Address:=17);
	ZTHL08	:	obj_ZTHL := (ID:=8, Address:=18);
	ZTHL09	:	obj_ZTHL := (ID:=9, Address:=19);
	ZTHL10	:	obj_ZTHL := (ID:=10, Address:=20);
	ZTHL11	:	obj_ZTHL := (ID:=11, Address:=21);
	ZTHL12	:	obj_ZTHL := (ID:=12, Address:=22);
	ZTHL13	:	obj_ZTHL := (ID:=13, Address:=23);



(*
	ZTHL10	:	obj_ZTHL := (ID:=4, Address:=14);  		(* ZTHL04 - CIR04  non montata *)
	ZTHL11	:	obj_ZTHL := (ID:=5, Address:=15);	 	(* ZTHL05 - CIR03  *)
	ZTHL12	:	obj_ZTHL := (ID:=3, Address:=3);
	ZTHL13	:	obj_ZTHL := (ID:=4, Address:=4);
	ZTHL14	:	obj_ZTHL := (ID:=5, Address:=5);
	ZTHL15	:	obj_ZTHL := (ID:=6, Address:=6);
	ZTHL16	:	obj_ZTHL := (ID:=7, Address:=7);
	ZTHL17	:	obj_ZTHL := (ID:=8, Address:=8);

	ZTHL19	:	obj_ZTHL := (ID:=10, Address:=10);


	ZTHL18	:	obj_ZTHL := (ID:=9, Address:=18); (* ZTHL08 *)
*)



	(** Communication **)
	(* ModBus *)
	MODB01	:	obj_MODBUS		:= (ID:=1, COM:=3, BAUDRATE:=BAUD_19200, RS485:=TRUE);
	MODB02	:	obj_MODBUS		:= (ID:=2, COM:=4, BAUDRATE:=BAUD_9600, RS485:=TRUE);
	MODB03	:	obj_MODBUS_TCP 	:= (ID:=1, IP:='192.168.100.4');

	(* M-Bus *)
	MBUS01	:	obj_MBUS		:= (ID:=1, COM:=2, BAUDRATE:=BAUD_2400);

	(**** SIMULATION ONLY ****)

	AggiornaLog: BOOL;

	(*...*)
END_VAR

(* Global variable list: LON/Module_1/InterfaceBlock_Module_1 *)
VAR_GLOBAL CONSTANT
(******************************************)
(* Automatic generated code, do not edit! *)
(******************************************)
	abSignature_Module_1 : ARRAY[0..15] OF BYTE := 16#69,16#29,16#EC,16#18,16#3D,16#49,16#AF,16#4B,16#92,16#46,16#53,16#8D,16#F7,16#9F,16#84,16#C4;
	wConfigSize_Module_1 : WORD := 541;
	abInterface_Module_1 : ARRAY[0..135] OF DWORD :=
		16#D028C1F1, 16#219F0D0A, 16#6041B800, 16#06246830, 16#428B2E71, 16#64B95263, 16#FE000902, 16#2A050140, 
		16#00284095, 16#B2680DFC, 16#1C383063, 16#80015566, 16#CCD57140, 16#491D7775, 16#D5B152C7, 16#31D509A2, 
		16#D48882D5, 16#B8C2D6F1, 16#58664BDA, 16#129C49F3, 16#B7137DBE, 16#334D42A4, 16#13284D97, 16#A11A9D0A, 
		16#EC5BB754, 16#8A7D5A96, 16#DDB165D5, 16#251B7427, 16#B7794192, 16#0B526EDD, 16#6DDBBE1D, 16#92AEDBB2, 
		16#E596450B, 16#2D4C8065, 16#4A4D6BD7, 16#D9BA71CB, 16#B041776E, 16#15932F4C, 16#77EA5BF9, 16#EBD20D4B, 
		16#C9946573, 16#4D6B747E, 16#16C4CAB2, 16#065A4DD9, 16#3BA926E5, 16#7AE06C0A, 16#73B4BD85, 16#AD820478, 
		16#18B1AF54, 16#10554D2A, 16#B6D25295, 16#3E949D0A, 16#86651B94, 16#C01B6DE5, 16#CB56AAD1, 16#C09794C8, 
		16#0E452A4F, 16#D3AF3187, 16#634B0254, 16#A9229B03, 16#0DDCB665, 16#5C248436, 16#0BB7EE54, 16#46A65682, 
		16#F2A2594E, 16#46D29A10, 16#66FA28DC, 16#031AE0B4, 16#24A2A921, 16#E8CEC315, 16#12B88A94, 16#B14105CA, 
		16#58F608DD, 16#D3BE851A, 16#92402D6E, 16#216A74A8, 16#EBB6A8CC, 16#19D88A0D, 16#D2518944, 16#B31095DE, 
		16#EBCE48AD, 16#49C33B55, 16#A7422F59, 16#F39AD2D0, 16#D53C3E25, 16#7572E178, 16#8A066673, 16#40F93B2B, 
		16#0418102A, 16#FF000702, 16#10B08496, 16#A168016C, 16#64610830, 16#D908B0E2, 16#F005E684, 16#AED89C34, 
		16#9D9C1307, 16#83007FD6, 16#008D4EA0, 16#C64EA28E, 16#E0890497, 16#C9241020, 16#1510A0E0, 16#E0D5E009, 
		16#9C223CA9, 16#53862716, 16#B87E21AE, 16#D6E27AA5, 16#AE678CEB, 16#07B98E39, 16#EB9AE43A, 16#51AE6F93, 
		16#7A67B9EE, 16#9AEB01E6, 16#2E6CAE7F, 16#E7FAD0B9, 16#1BA1EBC5, 16#BA7E8CAE, 16#89E93A51, 16#AE23A8EB, 
		16#C3BABEA8, 16#EB8DEB3A, 16#C4AE2BB0, 16#BA33BBFE, 16#00EB51ED, 16#201C8A4F, 16#BA8C0990, 16#82543B63, 
		16#71C0A0CC, 16#70A0C080, 16#D9A74C4B, 16#75D29E18, 16#1A95BCF4, 16#E7FB8DA7, 16#074A9CF0, 16#000000EC;
END_VAR

(* Global variable list: LON/Module_1/Runtime_Module_1 *)
VAR_GLOBAL
(******************************************)
(* Automatic generated code, do not edit! *)
(******************************************)
	mbxModule_1 : MBX_Full;
	InDataTelegram_Module_1 : ARRAY[0..255] OF BYTE;
	OutDataTelegram_Module_1 : ARRAY[0..511] OF BYTE;

	xInitRunning_Module_1 : BOOL := FALSE;
	unLastLen_mbxModule_1 : UINT;
END_VAR

(* Data type in LON/Enumerations *)
TYPE alarm_type_t :
(
	AL_HEADER := -13,
	AL_FOOTER := -12,
	AL_DEBUG := -11,
	AL_INFO := -10,
	AL_SYSTEM_INFO := -6,
	AL_VALUE_INVALID := -5,
	AL_CONSTANT := -4,
	AL_OFFLINE := -3,
	AL_UNKNOWN := -2,
	AL_NUL := -1,
	AL_NO_CONDITION := 0,
	AL_ALM_CONDITION := 1,
	AL_TOT_SVC_ALM_1 := 2,
	AL_TOT_SVC_ALM_2 := 3,
	AL_TOT_SVC_ALM_3 := 4,
	AL_LOW_LMT_CLR_1 := 5,
	AL_LOW_LMT_CLR_2 := 6,
	AL_HIGH_LMT_CLR_1 := 7,
	AL_HIGH_LMT_CLR_2 := 8,
	AL_LOW_LMT_ALM_1 := 9,
	AL_LOW_LMT_ALM_2 := 10,
	AL_HIGH_LMT_ALM_1 := 11,
	AL_HIGH_LMT_ALM_2 := 12,
	AL_FIR_ALM := 13,
	AL_FIR_PRE_ALM := 14,
	AL_FIR_TRBL := 15,
	AL_FIR_SUPV := 16,
	AL_FIR_TEST_ALM := 17,
	AL_FIR_TEST_PRE_ALM := 18,
	AL_FIR_ENVCOMP_MAX := 19,
	AL_FIR_MONITOR_COND := 20,
	AL_FIR_MAINT_ALERT := 21,
	AL_FATAL_ERROR := 30,
	AL_ERROR := 31,
	AL_WARNING := 32
);
END_TYPE

(* Data type in Logger *)
TYPE en_Logger_ErrLev :
(
	EL_Log			:=0,
	EL_Wrn			:=1,
	EL_Alarm		:=2,
	EL_AlarmStop	:=3
);
END_TYPE

(* Data type in Logger *)
TYPE en_Logger_Status :
(
	S_Logger_UNKNOWN := 0,
	S_Logger_IDLE,
	S_Logger_WAITCONN,
	S_Logger_WAITTX,
	S_Logger_WAITRESP,
	S_Logger_ERROR
);
END_TYPE

(* Data type *)
TYPE en_SYS_Objects :
(
	EO_SYS		:=0,  (* PLC *)
	EO_VPN		:=1,  (* VPN *)
	EO_DOOR		:=2,  (* Door & access control *)

	EO_CAL		:=10, (* Caldaia *)
	EO_CIR		:=11, (* Circolatore *)
	EO_CRON		:=12, (* Crono-termostato *)
	EO_VRD		:=13, (* Valvola miscelatore pannelli *)
	EO_CTL		:=14, (* Contalitri *)
	EO_CTB		:=15, (* Contabilizzatore *)
	EO_TPV		:=16, (* Temperature probes values *)
	EO_PPV		:=17, (* Pressure probes values *)
	EO_PBV		:=18, (* Over-Pressure Alarms *)
	EO_TBV		:=19, (* Over-Temperature Alarms *)
	EO_PMV		:=20, (* Under-Pressure Alarms *)
	EO_GRU		:=21, (* Gruppo termico *)
	EO_PDC		:=22, (* Pompa di calore *)
	EO_SOL		:=23, (* Pannello solare termico *)
	EO_ESOL		:=24, (* Pannello solare fotovoltaico *)
	EO_GAS		:=25, (* Contatore GAS *)
	EO_PORT		:=26, (* Misuratore di portata *)
	EO_FPV		:=27, (* Flow probes values *)
	EO_ANZ		:=28, (* Analizzatore di rete *)
	EO_SCA		:=29, (* Signal Control Alarms *)
	EO_LUX		:=30, (* Base Illumination point *)
	EO_LUXM		:=31, (* Metered Illumination point *)
	EO_PSG		:=32, (* Sensore di passaggio *)
	EO_HVAC		:=33, (* Heating, Ventilating and Air Conditioning *)
	EO_HYGRV	:=34, (* Relative Humidity sensors value *)
	EO_COOV		:=35, (* Carbon Dioxide CO2 sensors value *)
	EO_INV		:=36, (* Inverter *)
	EO_STR		:=37, (* Smart string box *)

	EO_CIRD		:=39, (* Double CIR *)
	EO_ACS		:=40, (* Hot domestic water *)
	EO_FRG		:=41, (* Frigo *)
	EO_THER		:=42, (* Thermostat *)
	EO_CIRM		:=43, (* Modbus CIR *)
	EO_CIRDM	:=44, (* Modbus double CIR *)

	EO_ZGW			:=200,  (* ZigBee - Gateway *)
	EO_ZRM			:=201,	(* ZigBee - Repeater *)
	EO_ZREL			:=202,	(* ZigBee - Actuator rele *)
	EO_ZTHL			:=203,	(* ZigBee - Temperature Sensor *)

	EO_ASGW			:=250,	(* ASi - Gateway *)
	EO_ASCBI		:=251,	(* ASi - Input Board, Ciabatta *)

	EO_LON			:=1000, (* Bus - LON *)
	EO_MODBUS		:=1001, (* Bus - MODBUS *)
	EO_MBUS			:=1002, (* Bus - M-BUS *)
	EO_MODBUS_TCP	:=1003, (* Bus - MODBUS TCP *)

	EO_GENERIC		:=9000, (* Generic dataset *)
	EO_EXPO			:=9001 (* EXPO dataset *)
);
END_TYPE

(* Data type *)
TYPE en_SYS_Status :
(
	S_UNKNOWN  := 0,
	S_STARTUP,
	S_INIT_RTC,
	S_INIT_VAR,
	S_AUTOTEST,
	S_RUNNING,
	S_SHUTDOWN,
	S_HALT
);
END_TYPE

(* Data type in LON/Enumerations *)
TYPE file_request_t :
(
	FR_NUL := -1,
	FR_OPEN_TO_SEND := 0,
	FR_OPEN_TO_RECEIVE := 1,
	FR_CLOSE_FILE := 2,
	FR_CLOSE_DELETE_FILE := 3,
	FR_DIRECTORY_LOOKUP := 4,
	FR_OPEN_TO_SEND_RA := 5,
	FR_OPEN_TO_RECEIVE_RA := 6
);
END_TYPE

(* Data type in LON/Enumerations *)
TYPE file_status_t :
(
	FS_NUL := -1,
	FS_XFER_OK := 0,
	FS_LOOKUP_OK := 1,
	FS_OPEN_FAIL := 2,
	FS_LOOKUP_ERR := 3,
	FS_XFER_UNDERWAY := 4,
	FS_IO_ERR := 5,
	FS_TIMEOUT_ERR := 6,
	FS_WINDOW_ERR := 7,
	FS_AUTH_ERR := 8,
	FS_ACCESS_UNAVAIL := 9,
	FS_SEEK_INVALID := 10,
	FS_SEEK_WAIT := 11
);
END_TYPE

(* Data type in LON/Enumerations *)
TYPE hvac_t :
(
	HVAC_NUL := -1,
	HVAC_AUTO := 0,
	HVAC_HEAT := 1,
	HVAC_MRNG_WRMUP := 2,
	HVAC_COOL := 3,
	HVAC_NIGHT_PURGE := 4,
	HVAC_PRE_COOL := 5,
	HVAC_OFF := 6,
	HVAC_TEST := 7,
	HVAC_EMERG_HEAT := 8,
	HVAC_FAN_ONLY := 9,
	HVAC_FREE_COOL := 10,
	HVAC_ICE := 11,
	HVAC_MAX_HEAT := 12,
	HVAC_ECONOMY := 13,
	HVAC_DEHUMID := 14,
	HVAC_CALIBRATE := 15,
	HVAC_EMERG_COOL := 16,
	HVAC_EMERG_STEAM := 17,
	HVAC_MAX_COOL := 18,
	HVAC_HVC_LOAD := 19,
	HVAC_NO_LOAD := 20
);
END_TYPE

(* Data type in LON/Enumerations *)
TYPE object_request_t :
(
	RQ_NUL := -1,
	RQ_NORMAL := 0,
	RQ_DISABLED := 1,
	RQ_UPDATE_STATUS := 2,
	RQ_SELF_TEST := 3,
	RQ_UPDATE_ALARM := 4,
	RQ_REPORT_MASK := 5,
	RQ_OVERRIDE := 6,
	RQ_ENABLE := 7,
	RQ_RMV_OVERRIDE := 8,
	RQ_CLEAR_STATUS := 9,
	RQ_CLEAR_ALARM := 10,
	RQ_ALARM_NOTIFY_ENABLED := 11,
	RQ_ALARM_NOTIFY_DISABLED := 12,
	RQ_MANUAL_CTRL := 13,
	RQ_REMOTE_CTRL := 14,
	RQ_PROGRAM := 15,
	RQ_CLEAR_RESET := 16,
	RQ_RESET := 17,
	RQ_CLEAR_LOG := 18,
	RQ_LOAD_PROGRAM := 19,
	RQ_RUN_PROGRAM := 20,
	RQ_HALT_PROGRAM := 21,
	RQ_RESTART_PROGRAM := 22,
	RQ_UNLOAD_PROGRAM := 23,
	RQ_STEP_PROGRAM := 24
);
END_TYPE

(* Data type in LON/Enumerations *)
TYPE priority_level_t :
(
	PR_NUL := -1,
	PR_LEVEL_0 := 0,
	PR_LEVEL_1 := 1,
	PR_LEVEL_2 := 2,
	PR_LEVEL_3 := 3,
	PR_1 := 4,
	PR_2 := 5,
	PR_3 := 6,
	PR_4 := 7,
	PR_6 := 8,
	PR_8 := 9,
	PR_10 := 10,
	PR_16 := 11
);
END_TYPE

(* Data type in Plant_Objects *)
TYPE typ_Clima : (* CURVA CLIMATICA *)
STRUCT
	InitOK:		BOOL;
	Points: 	ARRAY [0..10] OF POINT;
END_STRUCT
END_TYPE

(* Data type in Plant_Objects *)
TYPE typ_Cron_Calendar :
STRUCT
	Profile		: ARRAY[0..384] OF BYTE;
END_STRUCT
END_TYPE

(* Data type in Plant_Objects *)
TYPE typ_Cron_Jolly :
STRUCT
	Start		: DT;
	End			: DT;
	Temp		: WORD;
	Flags		: WORD; (* B0:Enabled B1..B15:Unused *)
END_STRUCT
END_TYPE

(* Data type in Plant_Objects *)
TYPE typ_Cron_Profile :
STRUCT
	Flags		: WORD;
	Setpoint	: ARRAY [0..95] OF WORD;
END_STRUCT
END_TYPE

(* Data type in Plant_Objects *)
TYPE typ_Frigo :
STRUCT
	Status	:	BOOL;		(* 0=OFF, 1=ON	*)
	Mode	:	BOOL;		(* 0=COLD, 1=HOT	*)
	Reset	:	BOOL;		(* 1=RESET	*)

	Alarm	:	DWORD;		(* 30 alarms of type bool grouped in one variable of 32 bits (last 2 don't used) *)

	(*  ALARM CODE (bit order of dword "Alarm": first is bit 0, last bit29)
        8	:	Allarme flussostato
		9	:	Allarme termica pompa condensante 
		10	:	Allarme termica pompa evaporante 
		11	:	Allarme resa 
		12	:	Allarme termica compressore circuito 1 
		13	:	Allarme bassa pressione circuito 1
		14	:	Allarme alta pressione circuito 1 
		15	:	Allarme antigelo circuito 1	
		16	:	Allarme termica ventilatore circuito 1	
		17	:	Allarme pressostato olio crcuito 1	
		18	:	Allarme sonda circuito 1	
		19	:	Allarme termica compressore circuito 2	
		20	:	Allarme bassa pressione circuito 2	
		21	:	Allarme alta pressione circuito 2	
		22	:	Allarme antigelo circuito 2	
		23	:	Allarme termica ventilatore circuito 2	
		24	:	Allarme pressostato olio circuito 2	
		25	:	Allarme sonda circuito 2	
		26	:	Allarme monitor tensione	
		27	:	Allarme pumpdown circuito 1	
		28	:	Allarme pumpdown circuito 2	
		29	:	Allarme eeprom	
		30	:	Allarme clock calendar	
		80	:	Allarme flussostato recuperatore	
		81	:	Allarme termica compressore circuito 1A	
		82	:	Allarme termica compressore circuito 1B	
		83	:	Allarme termica pompa evaporatore 1	
		84	:	Allarme termica pompa evaporatore 2	
		85	:	Allarme termica pompa evaporatore 3	
		86	:	Allarme antigelo evaporatore circuito 1	
		87	:	Allarme antigelo evaporatore circuito 2	
	*)


END_STRUCT
END_TYPE

(* Data type in Logger *)
TYPE typ_Logger :
STRUCT
	Status		: en_Logger_Status;

	SendReq		: BOOL;
	SendIdx		: DWORD;
	SendData	: ARRAY [0..MAX_SEND_TCP_CLIENT] OF BYTE;
	SendLen		: DINT;

	TData		: ARRAY [0..MAX_SEND_TCP_CLIENT] OF BYTE;
	TLen		: DINT;

	LastIdxPos	: DWORD;

	(* Temporary variables used by objects *)
	s1			: STRING(256);
	i1			: WORD;

END_STRUCT
END_TYPE

(* Data type in Plant_Objects *)
TYPE typ_MODBUS_CIR :
STRUCT
	PumpStatus		:	WORD;
	PumpFault		:	BOOL;
	PumpBoardTemp	:	INT;	(* Electonic board temperature  [°C] *)
	PumpVoltage		:	WORD;	(* Input voltage rms [V] *)
	PumpCurrent		:	WORD;	(* Output current [E-3 A]	*)
	PumpRPM			:	WORD;	(* Round per minute [rpm] *)
	PumpPower		:	WORD;	(* Power [W] *)
	PumpOpTime		:	DWORD;	(* Pump operating time [h] *)
	PumpHead		:	WORD;	(* [E-1 m] *)
	PumpFlow		:	WORD;	(* Extimated flow [E-1 m3/h] *)
	PumpLiqTemp		:	WORD;	(* Liquid temperature [°C] *)
	PumpAlarm		:	ARRAY [0..14] OF WORD;

END_STRUCT
END_TYPE

(* Data type in Plant_Objects *)
TYPE typ_MODBUS_VAR : (* Gestione parametri MODBUS *)
STRUCT
	SlaveAddress	: BYTE;
	FunCode			: BYTE;
	FunAddress		: WORD;
	Refresh_Time	: BYTE; (* 0:No refresh x:Refresh in seconds *)
	Refresh_Cnt		: BYTE; (* INTERNAL *)
	Variable		: POINTER TO WORD;
	Variable_Size	: BYTE;
	Variable_Mirror : WORD; (* INTERNAL [Force refresh on read variables when <>0] *)
END_STRUCT
END_TYPE

(* Data type *)
TYPE typ_SYS :
STRUCT
	Status			: en_SYS_Status;
	Warning			: BOOL;
	Alarm			: BOOL;
	AlarmStop		: BOOL;

	Time_LogString	: STRING;
	Time_Year		: WORD;
	Time_Month		: BYTE;
	Time_Day		: BYTE;
	Time_Hour		: BYTE;
	Time_Minute		: BYTE;

	Time_CT_DT		: DT;
	Time_CT_Day		: WORD;
	Time_CT_Quarter	: BYTE;

	LastLogs_Idx	: BYTE;
	LastLogs_Dat	: ARRAY[0..5] OF STRING;
	LastLogs_Msg	: ARRAY[0..5] OF STRING;

END_STRUCT
END_TYPE

(* Data type in Plant_Objects *)
TYPE typ_VisuStrutturaMbus :
STRUCT

	sdNodoPresente: STRING(16);
	sdEnergia: STRING(16);
	sdPotenza: STRING(16);
	sdVolume: STRING(16);
	sdFlow: STRING(16);
	sdTempIngresso: STRING(8);
	sdTempaUscita: STRING(8);
	sdTempDelta: STRING(8);

END_STRUCT
END_TYPE

(* Data type in LON/NetworkVariables *)
TYPE typSnvtAlarm : 
STRUCT
	abLocation : ARRAY[0..5] OF BYTE;
	wObjectId : WORD;
	bAlarmType : BYTE (* enum type alarm_type_t *);
	bPriorityLevel : BYTE (* enum type priority_level_t *);
	wIndexToSnvt : WORD;
	abValue : ARRAY[0..3] OF BYTE;
	wYear : WORD;
	bMonth : BYTE;
	bDay : BYTE;
	bHour : BYTE;
	bMinute : BYTE;
	bSecond : BYTE;
	wMillisecond : WORD;
	abAlarmLimit : ARRAY[0..3] OF BYTE;
	bStatusInformation : BYTE; (* bit allocation of bStatusInformation:
	bit 0: NVI update counter LSB
	bit 1: NVI update counter
	bit 2: NVI update counter
	bit 3: NVI update counter MSB
	bit 4: timeout for NVI occurs (MaxRcvTime expired)
	bit 5: reserved
	bit 6: reserved
	bit 7: force NVO update *)
	bInternalUseOnly : BYTE; (* Do not use this byte in your application! *)
END_STRUCT
END_TYPE

(* Data type in LON/NetworkVariables *)
TYPE typSnvtFilePos : 
STRUCT
	diRwPtr : DINT;
	wRwLength : WORD;
	bStatusInformation : BYTE; (* bit allocation of bStatusInformation:
	bit 0: NVI update counter LSB
	bit 1: NVI update counter
	bit 2: NVI update counter
	bit 3: NVI update counter MSB
	bit 4: timeout for NVI occurs (MaxRcvTime expired)
	bit 5: reserved
	bit 6: reserved
	bit 7: force NVO update *)
	bInternalUseOnly : BYTE; (* Do not use this byte in your application! *)
END_STRUCT
END_TYPE

(* Data type in LON/NetworkVariables *)
TYPE typSnvtFileReq : 
STRUCT
	bRequest : BYTE (* enum type file_request_t *);
	wIndex : WORD;
	wReceiveTimeout : WORD;
	abDestAddress : ARRAY[0..4] OF BYTE (* union declaration *);
	bAuthOn : BYTE;
	bPrioOn : BYTE;
	bStatusInformation : BYTE; (* bit allocation of bStatusInformation:
	bit 0: NVI update counter LSB
	bit 1: NVI update counter
	bit 2: NVI update counter
	bit 3: NVI update counter MSB
	bit 4: timeout for NVI occurs (MaxRcvTime expired)
	bit 5: reserved
	bit 6: reserved
	bit 7: force NVO update *)
	bInternalUseOnly : BYTE; (* Do not use this byte in your application! *)
END_STRUCT
END_TYPE

(* Data type in LON/NetworkVariables *)
TYPE typSnvtFileStatus : 
STRUCT
	bStatus : BYTE (* enum type file_status_t *);
	wNumberOfFiles : WORD;
	wSelectedFile : WORD;
	abAdr : ARRAY[0..21] OF BYTE (* union declaration *);
	bStatusInformation : BYTE; (* bit allocation of bStatusInformation:
	bit 0: NVI update counter LSB
	bit 1: NVI update counter
	bit 2: NVI update counter
	bit 3: NVI update counter MSB
	bit 4: timeout for NVI occurs (MaxRcvTime expired)
	bit 5: reserved
	bit 6: reserved
	bit 7: force NVO update *)
	bInternalUseOnly : BYTE; (* Do not use this byte in your application! *)
END_STRUCT
END_TYPE

(* Data type in LON/NetworkVariables *)
TYPE typSnvtHvacMode : 
STRUCT
	bSnvtHvacMode : BYTE (* enum type hvac_t *);
	bStatusInformation : BYTE; (* bit allocation of bStatusInformation:
	bit 0: NVI update counter LSB
	bit 1: NVI update counter
	bit 2: NVI update counter
	bit 3: NVI update counter MSB
	bit 4: timeout for NVI occurs (MaxRcvTime expired)
	bit 5: reserved
	bit 6: reserved
	bit 7: force NVO update *)
	bInternalUseOnly : BYTE; (* Do not use this byte in your application! *)
END_STRUCT
END_TYPE

(* Data type in LON/NetworkVariables *)
TYPE typSnvtObjRequest : 
STRUCT
	wObjectId : WORD;
	bObjectRequest : BYTE (* enum type object_request_t *);
	bStatusInformation : BYTE; (* bit allocation of bStatusInformation:
	bit 0: NVI update counter LSB
	bit 1: NVI update counter
	bit 2: NVI update counter
	bit 3: NVI update counter MSB
	bit 4: timeout for NVI occurs (MaxRcvTime expired)
	bit 5: reserved
	bit 6: reserved
	bit 7: force NVO update *)
	bInternalUseOnly : BYTE; (* Do not use this byte in your application! *)
END_STRUCT
END_TYPE

(* Data type in LON/NetworkVariables *)
TYPE typSnvtObjStatus : 
STRUCT
	wObjectId : WORD;
	bBitfieldByteOffset2 : BYTE (* bit field *);
	bBitfieldByteOffset3 : BYTE (* bit field *);
	bBitfieldByteOffset4 : BYTE (* bit field *);
	bBitfieldByteOffset5 : BYTE (* bit field *);
	bStatusInformation : BYTE; (* bit allocation of bStatusInformation:
	bit 0: NVI update counter LSB
	bit 1: NVI update counter
	bit 2: NVI update counter
	bit 3: NVI update counter MSB
	bit 4: timeout for NVI occurs (MaxRcvTime expired)
	bit 5: reserved
	bit 6: reserved
	bit 7: force NVO update *)
	bInternalUseOnly : BYTE; (* Do not use this byte in your application! *)
END_STRUCT
END_TYPE

(* Data type in LON/NetworkVariables *)
TYPE typSnvtState : 
STRUCT
	bBitfieldByteOffset0 : BYTE (* bit field *);
	bBitfieldByteOffset1 : BYTE (* bit field *);
	bStatusInformation : BYTE; (* bit allocation of bStatusInformation:
	bit 0: NVI update counter LSB
	bit 1: NVI update counter
	bit 2: NVI update counter
	bit 3: NVI update counter MSB
	bit 4: timeout for NVI occurs (MaxRcvTime expired)
	bit 5: reserved
	bit 6: reserved
	bit 7: force NVO update *)
	bInternalUseOnly : BYTE; (* Do not use this byte in your application! *)
END_STRUCT
END_TYPE

(* Data type in LON/NetworkVariables *)
TYPE typSnvtSwitch : 
STRUCT
	bValue : BYTE;
	siState : SINT;
	bStatusInformation : BYTE; (* bit allocation of bStatusInformation:
	bit 0: NVI update counter LSB
	bit 1: NVI update counter
	bit 2: NVI update counter
	bit 3: NVI update counter MSB
	bit 4: timeout for NVI occurs (MaxRcvTime expired)
	bit 5: reserved
	bit 6: reserved
	bit 7: force NVO update *)
	bInternalUseOnly : BYTE; (* Do not use this byte in your application! *)
END_STRUCT
END_TYPE

(* Data type in LON/NetworkVariables *)
TYPE typSnvtTempP : 
STRUCT
	iSnvtTempP : INT;
	bStatusInformation : BYTE; (* bit allocation of bStatusInformation:
	bit 0: NVI update counter LSB
	bit 1: NVI update counter
	bit 2: NVI update counter
	bit 3: NVI update counter MSB
	bit 4: timeout for NVI occurs (MaxRcvTime expired)
	bit 5: reserved
	bit 6: reserved
	bit 7: force NVO update *)
	bInternalUseOnly : BYTE; (* Do not use this byte in your application! *)
END_STRUCT
END_TYPE

(* Data type in LON/NetworkVariables *)
TYPE typSnvtTimeStamp : 
STRUCT
	iYear : INT;
	bMonth : BYTE;
	bDay : BYTE;
	bHour : BYTE;
	bMinute : BYTE;
	bSecond : BYTE;
	bStatusInformation : BYTE; (* bit allocation of bStatusInformation:
	bit 0: NVI update counter LSB
	bit 1: NVI update counter
	bit 2: NVI update counter
	bit 3: NVI update counter MSB
	bit 4: timeout for NVI occurs (MaxRcvTime expired)
	bit 5: reserved
	bit 6: reserved
	bit 7: force NVO update *)
	bInternalUseOnly : BYTE; (* Do not use this byte in your application! *)
END_STRUCT
END_TYPE

(* POU PLC_PRG, ST *)
PROGRAM PLC_PRG
VAR
	Timer1: TON; (* Fast controls tick *)
	Timer2: TON; (* Plant control tick *)
	Timer3: TON; (* Logger timer *)

	T_CIR01		:	INT;
	T_CIR02		:	INT;
	T_CIR03		:	INT;
	T_CIR04		:	INT;
	T_CIRD01	:	INT;
	T_CIRD02	:	INT;

	T_Valve01	:	INT;
	T_Valve02	:	INT;
	T_Valve03	:	INT;
	T_Valve04	:	INT;

	SecCircuitLogic	:	BOOL;	(* Secondary circuit request: LOGICAL ON/OFF *)
	SecCircuitReal	:	BOOL;	(* Secondart circuit request: REAL ON/OFF	 *)

	i : INT;

END_VAR
(******************************************************************************
 ****                           MAIN TASK CODE                             ****
 ******************************************************************************

	Network setup:
		IP  = 192.168.100.2 | MSK = 255.255.255.0
		GW	= 192.168.100.1 | DNS = 192.168.100.1
		SNTP = 193.204.114.232 (3600s) ==> 192.168.100.3

*)

(*==============================*)
(*===== Main status machine ====*)
(*==============================*)
Main_Stm();

(*==============================*)
(*== Running cycle operations ==*)
(*==============================*)
IF SYS.Status>S_INIT_VAR THEN
	(* Execute cycle processes *)
	(* Update LON output variables (needs to be here to obtain only one refresh) *)
	GRU01.Heartbeat( CLIM:=GRU01_Clima );
	(* Execute LON process *)
	Module_1_PRG();

	(* Count water pulses *)
	CTL01(CTL_ST:=CTL01_ST, COUNT:=Ctl01_Counter);
	CTL02(CTL_ST:=CTL02_ST, COUNT:=Ctl02_Counter);

	(* ModBus *)
	MODB01();

	CIR02(ModBus:=MODB01, Pump_AL:=NOT CIR02_AL, Pump_AUTO:=NOT CIR02_AUTO);
	CIR03(ModBus:=MODB01, Pump_AL:=NOT CIR03_AL, Pump_AUTO:=NOT CIR03_AUTO);
	CIR04(ModBus:=MODB01, Pump_AL:=NOT CIR04_AL, Pump_AUTO:=NOT CIR04_AUTO);

	MODB02();

	(*FRG01(ModBus:=MODB02);*)

	(* TCP ModBus *)
	MODB03();

	ZTHL01(MODBUS:=MODB03);
	ZTHL02(MODBUS:=MODB03);
	ZTHL03(MODBUS:=MODB03);
	ZTHL04(MODBUS:=MODB03);
(*	ZTHL05(MODBUS:=MODB03); *)
	ZTHL06(MODBUS:=MODB03);
	ZTHL07(MODBUS:=MODB03);
	ZTHL08(MODBUS:=MODB03);
	ZTHL09(MODBUS:=MODB03);
	ZTHL10(MODBUS:=MODB03);
	ZTHL11(MODBUS:=MODB03);
	ZTHL12(MODBUS:=MODB03);
	ZTHL13(MODBUS:=MODB03);


	(* M-Bus *)
	MBUS01();

	CTB01(MBUS:=MBUS01);

END_IF

(*==============================*)
(*== System cycle operations ===*)
(*==============================*)
(* Execute TCP processes *)
Logger_Proc();
Remote_Proc();
(* Update user led *)
USRLED_Update();
(* Execute Cron Editor commands *)
CronEd();

(* Environment temperature *)
IF NOT TPV01.ERR THEN T_AMB := S01;
ELSE T_AMB := Plant_DefaultTAmb;
END_IF


(**** SIMULATION ONLY ****)
(*...*)
END_PROGRAM
ACTION Main_Stm:
CASE Sys.Status OF

	S_STARTUP:
		Sys.Status:=S_INIT_RTC;

	S_INIT_RTC:
		(* Check RTC and update from network *)
		RTC_Update();
		(* Check time *)
		IF Sys.Time_Year>2000 THEN
			Sys.Status:=S_INIT_VAR;
		END_IF

	S_INIT_VAR:
		LogEv(EL_Wrn,EO_SYS,0,1,CONCAT('System_startup_v',WORD_TO_STRING(Plant_SW_VER)));
		Sys.Status:=S_RUNNING;

	S_RUNNING:
		Timer1(IN:=NOT Timer1.Q,PT:=T#50ms);
		IF Timer1.Q THEN
			(* Update meters *)

			(* Update system checks *)
			SYS_Proc();
		END_IF

		Timer2(IN:=NOT Timer2.Q,PT:=T#500ms);
		IF Timer2.Q THEN
			(* Read current date/time *)
			RTC_Update();


			(* Probes *)
			TPV01(IN:=S01);
			TPV02(IN:=S02);
			TPV03(IN:=S03);
			TPV04(IN:=S04);
			TPV05(IN:=S05);
			TPV06(IN:=S06);
			TPV07(IN:=S07);
			TPV08(IN:=S08);
			TPV09(IN:=S09);
			TPV04.Mean();
			TPV04(AVG=>FRG01.Twater_In);
			TPV05.Mean();
			TPV05(AVG=>FRG01.Twater_Out);


			(* Temperature *)
		(*	T_CIR01 := SEL(ZTHL04.ERR,ZTHL04.OUT_TEMP,Plant_DefaultTAmb); 	(* Sonda non presente *) *)
			T_CIR01 := Plant_DefaultTAmb; 		(* Sonda non presente Zona Custode *)


			(* Limito la lettura della sonda temperatura per evitare dissevizi *)
			T_CIR03 := SEL(ZTHL02.ERR,LIMIT(ZTHL02.OUT_TEMP,180,1000),Plant_DefaultTAmb);       (* Verifico che la minima non sia troppo minimo *)
			T_CIR03 := MIN (T_CIR03,SEL(ZTHL12.ERR,LIMIT(ZTHL12.OUT_TEMP,180,1000),Plant_DefaultTAmb)); (* Sonda Sala Brunelli CIRM02 *)

			(* Limito la lettura della sonda temperatura per evitare dissevizi *)
			T_CIR02 :=  SEL(ZTHL03.ERR,LIMIT(ZTHL03.OUT_TEMP,180,1000),Plant_DefaultTAmb);  	(* Sonda Ragioneria CIRM01 *)


			(* Limito la lettura della sonda temperatura per evitare dissevizi *)
			T_CIR04 := SEL(ZTHL01.ERR,LIMIT(ZTHL01.OUT_TEMP,180,1000),Plant_DefaultTAmb);		(* Sonda Zona Vigili PT P1 P2 *)
			T_CIR04 := MIN (T_CIR04,SEL(ZTHL07.ERR,LIMIT(ZTHL07.OUT_TEMP,180,1000),Plant_DefaultTAmb));
			T_CIR04 := MIN (T_CIR04,SEL(ZTHL06.ERR,LIMIT(ZTHL06.OUT_TEMP,180,1000),Plant_DefaultTAmb));
			T_CIR04 := MIN (T_CIR04,SEL(ZTHL11.ERR,LIMIT(ZTHL11.OUT_TEMP,180,1000),Plant_DefaultTAmb));

			(* Limito la lettura della sonda temperatura per evitare dissevizi *)
			T_CIRD01 := SEL(ZTHL08.ERR,LIMIT(ZTHL08.OUT_TEMP,180,1000),Plant_DefaultTAmb);		(* Sonda Zona Nuova FC P1 P2 P3 *)
			T_CIRD01 := MIN (T_CIRD01,SEL(ZTHL09.ERR,LIMIT(ZTHL09.OUT_TEMP,180,1000),Plant_DefaultTAmb));
			T_CIRD01 := MIN (T_CIRD01,SEL(ZTHL10.ERR,LIMIT(ZTHL10.OUT_TEMP,180,1000),Plant_DefaultTAmb));
			T_CIRD01 := MIN (T_CIRD01,SEL(ZTHL13.ERR,LIMIT(ZTHL13.OUT_TEMP,180,1000),Plant_DefaultTAmb));


			(* Limito la lettura della sonda temperatura per evitare dissevizi *)
			T_CIRD02 :=  SEL(ZTHL04.ERR,LIMIT(ZTHL04.OUT_TEMP,180,1000),Plant_DefaultTAmb);  	(* Sonda Zona Nuova Fan Coil CIRD02 *)

			(* Thermostats *)
			THER01(Temperature:=T_CIR01, Run=>CIR01.OnOff);(*, AntifreezeForce=>CIR01.CIR_RUN_REQ);*) (*Zona Custode *)
			THER02(Temperature:=T_CIR02, Run=>CIR02.OnOff);(*, AntifreezeForce=>CIR02.CIR_RUN_REQ);*)
			THER03(Temperature:=T_CIR03, Run=>CIR03.OnOff);(*, AntifreezeForce=>CIR03.CIR_RUN_REQ);*)
			THER04(Temperature:=T_CIR04, Run=>CIR04.OnOff);(*, AntifreezeForce=>CIR04.CIR_RUN_REQ);*)
			THER05(Temperature:=T_CIRD01, Run=>CIRD01.OnOff);(*, AntifreezeForce=>CIRD01.CIR_RUN_REQ);*)
			THER06(Temperature:=T_CIRD02, Run=>CIRD02.OnOff);(*, AntifreezeForce=>CIRD02.CIR_RUN_REQ);*)

			CRON01(SetPoint=>FRG01.SetPoint);

			(* CIR *)
			CIR01(Pump_AL:=NOT CIR01_AL, Pump_ST:=CIR01_ST, Pump_AUTO:=NOT CIR01_AUTO, CIR_EN=>CIR01_EN);

			CIR05(Pump_AL:=NOT CIR05_AL, Pump_AUTO:=NOT CIR05_AUTO, Tprobe:=TPV04.AVG, CIR_EN=>CIR05_EN, OnOff:=FRG01.Run);

			(* Double CIR *)
			CIRD01(PumpA_AL:=NOT CIRD01_A_AL, PumpB_AL:=NOT CIRD01_B_AL, PumpA_AUTO:=NOT CIRD01_A_AUTO, PumpB_AUTO:=NOT CIRD01_B_AUTO,
				   PumpA_En=>CIRD01_A_EN, PumpB_En=>CIRD01_B_EN);
			CIRD02(PumpA_AL:=NOT CIRD02_A_AL, PumpB_AL:=NOT CIRD02_B_AL, PumpA_AUTO:=NOT CIRD02_A_AUTO, PumpB_AUTO:=NOT CIRD02_B_AUTO,
				   PumpA_En=>CIRD02_A_EN, PumpB_En=>CIRD02_B_EN);

			(* Valves *)
			TPV06.Mean();
			T_Valve01 := SEL(TPV06.ERR,TPV06.AVG,Plant_VRD_TDefault);

			TPV07.Mean();
			T_Valve02 := SEL(TPV07.ERR,TPV07.AVG,Plant_VRD_TDefault);

			TPV08.Mean();
			T_Valve03 := SEL(TPV08.ERR,TPV08.AVG,Plant_VRD_TDefault);

			TPV09.Mean();
			T_Valve04 := SEL(TPV09.ERR,TPV09.AVG,Plant_VRD_TDefault);

			VRD02(RUN:=CIR02.Run, CLIM:=VRD02_Clima, TEMP:=T_Valve02, STATUS:=VRD02_ST, OUT_CL=>VRD02_CL, OUT_OP=>VRD02_OP);
			VRD01(RUN:=(CIR01.Run OR CIR02.Run), CLIM:=VRD01_Clima, TEMP:=T_Valve01, STATUS:=VRD01_ST, OUT=>VRD01_CTRL); (* Guasta *)
			VRD03(RUN:=CIR03.Run, CLIM:=VRD03_Clima, TEMP:=T_Valve03, STATUS:=VRD03_ST, OUT=>VRD03_CTRL);
			VRD04(RUN:=CIR04.Run, CLIM:=VRD04_Clima, TEMP:=T_Valve04, STATUS:=VRD04_ST, OUT=>VRD04_CTRL);				 (* Guasta *)




			(* Secondary circuit heat request *)
			SecCircuitLogic := CIR01.Ctrl_Run OR CIR02.Ctrl_Run OR CIR03.Ctrl_Run OR CIR04.Ctrl_Run OR CIRD01.Ctrl_Run OR CIRD02.Ctrl_Run;
			SecCircuitReal := CIR01.Run OR CIR02.Run OR CIR03.Run OR CIR04.Run OR CIRD01.Run OR CIRD02.Run;

			(* No secondary circuit heat request -->> Switch off immediatly CAL
			   Secondary circuit heat request -->> First switch on primary pump CIR01, when enabled switch on CAL *)
			GRU01.Run := SEL(SecCircuitLogic,FALSE,TRUE) AND SYS.AlarmStop=FALSE;


			(* Scrivo il setpoint in funzione della curva cliamatica più alta *)

			GRU01.SetPointManuale:=GRU01.Curve_Temp - GRU01.OffsetSetPointManuale;
			GRU01.SetPointManuale:=MAX(GRU01.SetPointManuale,SEL(VRD01.RUN,0,VRD01.Ctrl_SetPoint));
			GRU01.SetPointManuale:=MAX(GRU01.SetPointManuale,SEL(VRD02.RUN,0,VRD02.Ctrl_SetPoint));
			GRU01.SetPointManuale:=MAX(GRU01.SetPointManuale,SEL(VRD03.RUN,0,VRD03.Ctrl_SetPoint));
			GRU01.SetPointManuale:=MAX(GRU01.SetPointManuale,SEL(VRD04.RUN,0,VRD04.Ctrl_SetPoint));

			GRU01(CLIM:=GRU01_Clima,AbilitaSetPointManuale:=TRUE);




			(* Check plant status *)
			Lamp();

			(* Test toggle *)
			(*IF TEST1 THEN TEST1:=FALSE; ELSE TEST1:=TRUE; END_IF*)
		END_IF

		Timer3(IN:=NOT Timer3.Q,PT:=T#5m);
		IF Timer3.Q OR AggiornaLog THEN
			(* Trig logger *)
			LogTrig();
			(* Execute temporary CSV logger *)
			(*CSV_Log();*)
		END_IF

	S_SHUTDOWN:
		(* Stop sistema *)
		Sys.Status:=S_STARTUP;

	S_HALT:
		(* Aspetta uscita manuale *)
		Sys.Status:=S_STARTUP;

ELSE
	Sys.Status:=S_STARTUP;
END_CASE;
END_ACTION

(* POU LON/Module_1/Module_1_PRG, FBD *)
PROGRAM Module_1_PRG
VAR
	(* Automatic added code, do not change! *)
	LonMaster : Module_1_LonMaster;
	SFPTnodeObject : Module_1_SFPTnodeObject;
	Virtualfunctionalblock : Module_1_Virtualfunctionalblock;

	InData_LON AT %IB0 : ARRAY[0..23] OF BYTE;
	OutData_LON AT %QB0 : ARRAY[0..23] OF BYTE;
	(***** End of automatic added code. *****)

	(* Add your code here. *)
	LonState: BOOL;
	LonReset: BOOL;

END_VAR
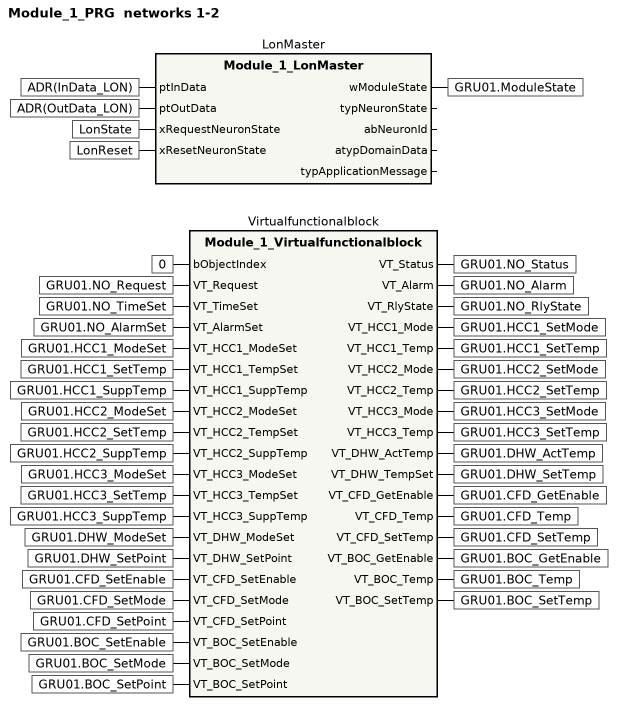
_FBD_ (* Function Block Diagram *)
NETWORK 1 (* Added by code generator *)
	LonMaster:Module_1_LonMaster(ptInData: ADR(InData_LON), ptOutData: ADR(OutData_LON), xRequestNeuronState: LonState, xResetNeuronState: LonReset) => GRU01.ModuleState
NETWORK 2
	Virtualfunctionalblock:Module_1_Virtualfunctionalblock(bObjectIndex: 0, VT_Request: GRU01.NO_Request, VT_TimeSet: GRU01.NO_TimeSet, VT_AlarmSet: GRU01.NO_AlarmSet, VT_HCC1_ModeSet: GRU01.HCC1_ModeSet, VT_HCC1_TempSet: GRU01.HCC1_SetTemp, VT_HCC1_SuppTemp: GRU01.HCC1_SuppTemp, VT_HCC2_ModeSet: GRU01.HCC2_ModeSet, VT_HCC2_TempSet: GRU01.HCC2_SetTemp, VT_HCC2_SuppTemp: GRU01.HCC2_SuppTemp, VT_HCC3_ModeSet: GRU01.HCC3_ModeSet, VT_HCC3_TempSet: GRU01.HCC3_SetTemp, VT_HCC3_SuppTemp: GRU01.HCC3_SuppTemp, VT_DHW_ModeSet: GRU01.DHW_ModeSet, VT_DHW_SetPoint: GRU01.DHW_SetPoint, VT_CFD_SetEnable: GRU01.CFD_SetEnable, VT_CFD_SetMode: GRU01.CFD_SetMode, VT_CFD_SetPoint: GRU01.CFD_SetPoint, VT_BOC_SetEnable: GRU01.BOC_SetEnable, VT_BOC_SetMode: GRU01.BOC_SetMode, VT_BOC_SetPoint: GRU01.BOC_SetPoint, VT_Alarm => GRU01.NO_Alarm, VT_RlyState => GRU01.NO_RlyState, VT_HCC1_Mode => GRU01.HCC1_SetMode, VT_HCC1_Temp => GRU01.HCC1_SetTemp, VT_HCC2_Mode => GRU01.HCC2_SetMode, VT_HCC2_Temp => GRU01.HCC2_SetTemp, VT_HCC3_Mode => GRU01.HCC3_SetMode, VT_HCC3_Temp => GRU01.HCC3_SetTemp, VT_DHW_ActTemp => GRU01.DHW_ActTemp, VT_DHW_TempSet => GRU01.DHW_SetTemp, VT_CFD_GetEnable => GRU01.CFD_GetEnable, VT_CFD_Temp => GRU01.CFD_Temp, VT_CFD_SetTemp => GRU01.CFD_SetTemp, VT_BOC_GetEnable => GRU01.BOC_GetEnable, VT_BOC_Temp => GRU01.BOC_Temp, VT_BOC_SetTemp => GRU01.BOC_SetTemp) => GRU01.NO_Status
_END_FBD_
(* the same logic as Structured Text *)
(* Network 1: Added by code generator *)
LonMaster(ptInData := ADR(InData_LON), ptOutData := ADR(OutData_LON), xRequestNeuronState := LonState, xResetNeuronState := LonReset);
GRU01.ModuleState := LonMaster.wModuleState;
(* Network 2 *)
Virtualfunctionalblock(bObjectIndex := 0, VT_Request := GRU01.NO_Request, VT_TimeSet := GRU01.NO_TimeSet, VT_AlarmSet := GRU01.NO_AlarmSet, VT_HCC1_ModeSet := GRU01.HCC1_ModeSet, VT_HCC1_TempSet := GRU01.HCC1_SetTemp, VT_HCC1_SuppTemp := GRU01.HCC1_SuppTemp, VT_HCC2_ModeSet := GRU01.HCC2_ModeSet, VT_HCC2_TempSet := GRU01.HCC2_SetTemp, VT_HCC2_SuppTemp := GRU01.HCC2_SuppTemp, VT_HCC3_ModeSet := GRU01.HCC3_ModeSet, VT_HCC3_TempSet := GRU01.HCC3_SetTemp, VT_HCC3_SuppTemp := GRU01.HCC3_SuppTemp, VT_DHW_ModeSet := GRU01.DHW_ModeSet, VT_DHW_SetPoint := GRU01.DHW_SetPoint, VT_CFD_SetEnable := GRU01.CFD_SetEnable, VT_CFD_SetMode := GRU01.CFD_SetMode, VT_CFD_SetPoint := GRU01.CFD_SetPoint, VT_BOC_SetEnable := GRU01.BOC_SetEnable, VT_BOC_SetMode := GRU01.BOC_SetMode, VT_BOC_SetPoint := GRU01.BOC_SetPoint);
GRU01.NO_Alarm := Virtualfunctionalblock.VT_Alarm;
GRU01.NO_RlyState := Virtualfunctionalblock.VT_RlyState;
GRU01.HCC1_SetMode := Virtualfunctionalblock.VT_HCC1_Mode;
GRU01.HCC1_SetTemp := Virtualfunctionalblock.VT_HCC1_Temp;
GRU01.HCC2_SetMode := Virtualfunctionalblock.VT_HCC2_Mode;
GRU01.HCC2_SetTemp := Virtualfunctionalblock.VT_HCC2_Temp;
GRU01.HCC3_SetMode := Virtualfunctionalblock.VT_HCC3_Mode;
GRU01.HCC3_SetTemp := Virtualfunctionalblock.VT_HCC3_Temp;
GRU01.DHW_ActTemp := Virtualfunctionalblock.VT_DHW_ActTemp;
GRU01.DHW_SetTemp := Virtualfunctionalblock.VT_DHW_TempSet;
GRU01.CFD_GetEnable := Virtualfunctionalblock.VT_CFD_GetEnable;
GRU01.CFD_Temp := Virtualfunctionalblock.VT_CFD_Temp;
GRU01.CFD_SetTemp := Virtualfunctionalblock.VT_CFD_SetTemp;
GRU01.BOC_GetEnable := Virtualfunctionalblock.VT_BOC_GetEnable;
GRU01.BOC_Temp := Virtualfunctionalblock.VT_BOC_Temp;
GRU01.BOC_SetTemp := Virtualfunctionalblock.VT_BOC_SetTemp;
GRU01.NO_Status := Virtualfunctionalblock.VT_Status;
END_PROGRAM

(* POU LON/Module_1/Master/Module_1_LonMaster, ST *)
FUNCTION_BLOCK Module_1_LonMaster
(******************************************)
(* Automatic generated code, do not edit! *)
(******************************************)
VAR_INPUT
	ptInData  : POINTER TO BYTE;
	ptOutData : POINTER TO BYTE;
	xRequestNeuronState : BOOL;
	xResetNeuronState : BOOL;
END_VAR
VAR_OUTPUT
	wModuleState : WORD; (* bit coded wModuleState:
	15: communication to I/O-module interrupted (error)
	14 - 08: reserved
	07: ready for Neuron initialization
	06: Neuron active
	05: user interface active
	04: internal module communication interrupted (error)
	03: CP synchronization running
	02: Neuron is configured online
	01 - 00: reserved *)

	typNeuronState : NeuronState;
	abNeuronId : ARRAY[0..5] OF BYTE;
	atypDomainData : ARRAY[0..1] OF DomainData;
	typApplicationMessage : ApplicationMessageData;
END_VAR
VAR
	bInternalCode : BYTE;
	bNvIndex : BYTE;
	wCpIndex : WORD;
	lonCom : FbLonBasicCommunication;

	xInitIsStarted : BOOL := FALSE;

	TimeoutTimer : TON;
	timeOutTime : TIME := T#1000ms;
	xStateMachineIsChecked : BOOL;
	xTimerStart : BOOL;

	iDomainTable : INT;
	xSendRequestPending : BOOL;
	trigRequest : R_TRIG;
	trigReset : R_TRIG;

	abMbxRxPrio0Buf: ARRAY [0..309] OF BYTE;
	abMbxRxPrio1Buf: ARRAY [0..517] OF BYTE;
	aMbxRxBufSize: ARRAY [0..1] OF UINT := 310, 518;
	aMbxRxBufList: ARRAY [0..1] OF POINTER TO BYTE;
	afbMbxRxFb: ARRAY [0..1] OF MBX2_RX_DEFRAG;
	astMbxRxCtx: ARRAY [0..1] OF stMbx2DefragContext;

	abMbxTxPrio0Buf: ARRAY [0..309] OF BYTE;
	abMbxTxPrio1Buf: ARRAY [0..517] OF BYTE;
	aMbxTxBufSize: ARRAY [0..1] OF UINT := 310, 518;
	aMbxTxBufList: ARRAY [0..1] OF POINTER TO BYTE;
	afbMbxTxFb: ARRAY [0..1] OF MBX2_TX_FRAG;

	astMbxTrackContext: ARRAY [0..0] OF stMbx2TrackContext;
END_VAR
VAR CONSTANT
END_VAR
aMbxRxBufList[0] := ADR(abMbxRxPrio0Buf[0]);
aMbxRxBufList[1] := ADR(abMbxRxPrio1Buf[0]);

aMbxTxBufList[0] := ADR(abMbxTxPrio0Buf[0]);
aMbxTxBufList[1] := ADR(abMbxTxPrio1Buf[0]);

mbxModule_1.Ressources.pDefragBufList := ADR(aMbxRxBufList);
mbxModule_1.Ressources.pDefragBufSizeList := ADR(aMbxRxBufSize);
mbxModule_1.Ressources.pDefragCtxPtrList := ADR(astMbxRxCtx);
mbxModule_1.Ressources.pDefragFbList := ADR(afbMbxRxFb);
mbxModule_1.Ressources.pFragBufList := ADR(aMbxTxBufList);
mbxModule_1.Ressources.pFragBufSizeList := ADR(aMbxTxBufSize);
mbxModule_1.Ressources.pFragFbList := ADR(afbMbxTxFb);

mbxModule_1.Ressources.unMaxAvailableRxPrioIndex := 1;
mbxModule_1.Ressources.unMaxAvailableTxPrioIndex := 1;

mbxModule_1.Ressources.pTrackStList := ADR(astMbxTrackContext);
mbxModule_1.Ressources.unMaxAvailableTrackIndex := 0;

mbxModule_1.Ressources.pabRxWin := ptInData + 1;
mbxModule_1.Ressources.pabTxWin := ptOutData + 1;
mbxModule_1.Ressources.bTxWinSize := 23;
mbxModule_1.Ressources.bRxWinSize := 23;

IF (mbxModule_1.bStatus.2 = TRUE) OR (mbxModule_1.bStatus.1 = TRUE) THEN
	mbxModule_1.MBX_RESET();
	xInitRunning_Module_1 := TRUE;
	xInitIsStarted := FALSE;
END_IF
mbxModule_1.MBX_CYCLE();

IF (mbxModule_1.bStatus.0 <> TRUE) THEN 
	wModuleState := 16#8000;
	RETURN;
ELSE
	wModuleState.15 := FALSE;
END_IF

xStateMachineIsChecked := FALSE;
IF xInitRunning_Module_1 = TRUE THEN
	IF xInitIsStarted = FALSE THEN
		SetParameter();
		lonCom.eInitState := INIT_SND_SGNTR_REQ;
		lonCom.CheckInitState();
		xInitIsStarted := TRUE;
		xStateMachineIsChecked := TRUE;
	END_IF
END_IF

typApplicationMessage.xMsgRcvd := FALSE;
typApplicationMessage.xRspRcvd := FALSE;
ResetNviUpdate();
WHILE (mbxModule_1.xRxPending) DO
	unLastLen_mbxModule_1 := mbxModule_1.unRxLen;
	mbxModule_1.pbRxData := ADR(InDataTelegram_Module_1);
	mbxModule_1.MBX_RETRIEVE();
	IF (mbxModule_1.nError <> MBX_OK) THEN EXIT; END_IF;
	bInternalCode := InDataTelegram_Module_1[0];

	IF (xInitRunning_Module_1 = TRUE) AND (lonCom.eInitState <> INIT_TRANSFER_CFG) THEN
		IF (FuCheckForValidInitCode(bInternalCode)) THEN
			SetParameter();
			lonCom.unLastLen := unLastLen_mbxModule_1;
			lonCom.CheckInitState();
			xInitRunning_Module_1 := NOT lonCom.xInitDone;
			xStateMachineIsChecked := TRUE;
		END_IF
	END_IF

	IF (bInternalCode = M2C_NVI_UPDT_OCCD) OR (bInternalCode = M2C_NV_VALUE_RSP) OR (bInternalCode = M2C_NVI_UPDT_TOUT) THEN
		bNvIndex := InDataTelegram_Module_1[1];
		CASE bNvIndex OF
			0, 2, 4: Module_1_PRG.SFPTnodeObject.DataReceived();
			6, 8, 10, 12, 14, 17, 19, 22, 24, 27, 29, 31, 33, 35, 37, 39, 41: Module_1_PRG.Virtualfunctionalblock.DataReceived();

		END_CASE;
	ELSIF (bInternalCode = M2C_CP_VALUE_RSP) THEN
		wCpIndex := InDataTelegram_Module_1[1] OR (InDataTelegram_Module_1[2] * 256);
		CASE wCpIndex OF

		END_CASE;
	ELSIF (bInternalCode = M2C_LON_MSG_RCVD) OR (bInternalCode = M2C_LON_RSP_RCVD) THEN
		ApplMsgReceived();
	ELSIF (bInternalCode = M2C_STATUS_RSP) THEN
		wModuleState := (wModuleState AND 16#FF00) + InDataTelegram_Module_1[1];
	ELSIF (bInternalCode = M2C_NEURON_ID) THEN
		FuMemCopy(ADR(InDataTelegram_Module_1[1]), ADR(abNeuronId), 6);
	ELSIF (bInternalCode = M2C_DOMAIN_DATA) THEN
		DomainDataRcvd();
	ELSIF (bInternalCode = M2C_MICRO_SERVER_STATUS_RSP) THEN
		NeuronStateRcvd();
	END_IF
END_WHILE

IF (xInitRunning_Module_1 = TRUE) AND ((lonCom.xCallStateMachine = TRUE) OR (TimeoutTimer.Q = TRUE)) AND (NOT xStateMachineIsChecked) THEN
	SetParameter();
	lonCom.xTimeOut := TimeoutTimer.Q;
	lonCom.CheckInitState();
END_IF
TimeoutTimer(IN:=lonCom.xTimerStart, PT:=timeOutTime);

trigRequest(CLK := xRequestNeuronState);
trigReset(CLK := xResetNeuronState);
IF (trigRequest.Q OR trigReset.Q) THEN
	RequestNeuronState();
END_IF
END_FUNCTION_BLOCK
ACTION ApplMsgReceived:
IF (InDataTelegram_Module_1[0] = M2C_LON_MSG_RCVD) THEN
	typApplicationMessage.typService := InDataTelegram_Module_1[1] AND 16#30;
	typApplicationMessage.bSourceSubnetId := InDataTelegram_Module_1[2];
	typApplicationMessage.bSourceNodeId := InDataTelegram_Module_1[3];
	typApplicationMessage.bCorrelator := InDataTelegram_Module_1[4];
	typApplicationMessage.bCode :=  InDataTelegram_Module_1[5];
	typApplicationMessage.bDataLength := UINT_TO_BYTE(unLastLen_mbxModule_1 - 6);
	IF typApplicationMessage.bDataLength > 48 THEN typApplicationMessage.bDataLength := 48; END_IF;
	FuMemSet(ADR(typApplicationMessage.abData), 0, SIZEOF(typApplicationMessage.abData));
	IF typApplicationMessage.bDataLength > 0 THEN
		FuMemCopy(ADR(InDataTelegram_Module_1[6]), ADR(typApplicationMessage.abData), typApplicationMessage.bDataLength);
	END_IF
	typApplicationMessage.xMsgRcvd := TRUE;
ELSE
	typApplicationMessage.typService := LON_RESPONSE;
	typApplicationMessage.bSourceSubnetId := InDataTelegram_Module_1[1];
	typApplicationMessage.bSourceNodeId := InDataTelegram_Module_1[2];
	typApplicationMessage.bCorrelator := 0;
	typApplicationMessage.bCode :=  InDataTelegram_Module_1[3];
	typApplicationMessage.bDataLength := UINT_TO_BYTE(unLastLen_mbxModule_1 - 4);
	IF typApplicationMessage.bDataLength > 48 THEN typApplicationMessage.bDataLength := 48; END_IF;
	FuMemSet(ADR(typApplicationMessage.abData), 0, SIZEOF(typApplicationMessage.abData));
	IF typApplicationMessage.bDataLength > 0 THEN
		FuMemCopy(ADR(InDataTelegram_Module_1[4]), ADR(typApplicationMessage.abData), typApplicationMessage.bDataLength);
	END_IF
	typApplicationMessage.xRspRcvd := TRUE;
END_IF
END_ACTION
ACTION DomainDataRcvd:
IF (unLastLen_mbxModule_1 = 17) THEN
	iDomainTable := InDataTelegram_Module_1[1];
	IF (iDomainTable < 0) OR (iDomainTable > 1) THEN RETURN; END_IF
	FuMemCopy(ADR(InDataTelegram_Module_1[2]), ADR(atypDomainData[iDomainTable].abDomainId), 6);
	atypDomainData[iDomainTable].bSubnet := InDataTelegram_Module_1[8];
	atypDomainData[iDomainTable].xIsNonClone := InDataTelegram_Module_1[9].7;
	atypDomainData[iDomainTable].bNodeId := InDataTelegram_Module_1[9] AND 16#7F;
	atypDomainData[iDomainTable].xIsInvalid := InDataTelegram_Module_1[10].7;
	atypDomainData[iDomainTable].bDomainIdLength := InDataTelegram_Module_1[10] AND 16#7F;
	FuMemCopy(ADR(InDataTelegram_Module_1[11]), ADR(atypDomainData[iDomainTable].abAuthenticationKey), 6);
END_IF
END_ACTION
ACTION NeuronStateRcvd:
IF (unLastLen_mbxModule_1 = 16) THEN
	typNeuronState.wCrcError := InDataTelegram_Module_1[1] + InDataTelegram_Module_1[2] * 256;
	typNeuronState.wTransactionTimeouts := InDataTelegram_Module_1[3] + InDataTelegram_Module_1[4] * 256;
	typNeuronState.wReceiveTransactionBuffersFull := InDataTelegram_Module_1[5] + InDataTelegram_Module_1[6] * 256;
	typNeuronState.wLostMessages := InDataTelegram_Module_1[7] + InDataTelegram_Module_1[8] * 256;
	typNeuronState.wMissedMessages := InDataTelegram_Module_1[9] + InDataTelegram_Module_1[10] * 256;
	typNeuronState.bResetCause := InDataTelegram_Module_1[11];
	typNeuronState.bNodeState := InDataTelegram_Module_1[12];
	typNeuronState.bFirmwareVersion := InDataTelegram_Module_1[13];
	typNeuronState.bLastErrorLogged := InDataTelegram_Module_1[14];
	typNeuronState.bModelNumber := InDataTelegram_Module_1[15];
END_IF
END_ACTION
ACTION RequestNeuronState:
OutDataTelegram_Module_1[0] := C2M_MICRO_SERVER_STATUS_QRY;
OutDataTelegram_Module_1[1] := BOOL_TO_BYTE(trigReset.Q);

mbxModule_1.bTxPrio := 1;
mbxModule_1.bTxProtID := 0;
mbxModule_1.pbTxData := ADR(OutDataTelegram_Module_1);
mbxModule_1.unTxLen := 2;
mbxModule_1.MBX_SEND();

IF (mbxModule_1.nError <> MBX_OK) THEN
	RETURN;
END_IF
END_ACTION
ACTION ResetNviUpdate:
Module_1_PRG.SFPTnodeObject.ResetNviUpdate();
Module_1_PRG.Virtualfunctionalblock.ResetNviUpdate();
END_ACTION
ACTION SetParameter:
lonCom.pMbx 			:= ADR(mbxModule_1);
lonCom.pInData 			:= ADR(InDataTelegram_Module_1);
lonCom.pOutData 		:= ADR(OutDataTelegram_Module_1);
lonCom.pTimer			:= ADR(TimeoutTimer);

lonCom.pActualSignature	:= ADR(abSignature_Module_1);
lonCom.pConfigBlock := ADR(abInterface_Module_1);
lonCom.wConfigSize 		:= wConfigSize_Module_1;
END_ACTION

(* POU LON/Module_1/NV_Interface/Module_1_SFPTnodeObject, ST *)
FUNCTION_BLOCK Module_1_SFPTnodeObject
(******************************************)
(* Automatic generated code, do not edit! *)
(******************************************)
VAR_INPUT
	bObjectIndex : BYTE := 0;
	nvoStatus : typSnvtObjStatus;
	nvoFileStat : typSnvtFileStatus;

END_VAR
VAR_OUTPUT
	nviRequest : typSnvtObjRequest;
	nviFileReq : typSnvtFileReq;
	nviFilePos : typSnvtFilePos;

END_VAR
VAR
	xSetOnce : BOOL := TRUE;
	xDataInUpdated : BOOL := FALSE;
	nvoStatusLast: typSnvtObjStatus;
	nvoFileStatLast: typSnvtFileStatus;

	cmd : BYTE;
	z : INT;
	bNvRelativeIdx : BYTE;
	bNvAbsoluteIdx : BYTE;
	wCpRelativeIdx : WORD;
	wCpAbsoluteIdx : WORD;
END_VAR
VAR CONSTANT
	bNvStartIndex : BYTE := 0;
	wCpStartIndex : WORD := 65535;
	bLmoCount : BYTE := 1;
END_VAR
IF (xInitRunning_Module_1 = TRUE) AND (xSetOnce = TRUE) THEN
	xSetOnce := FALSE;
	CachePointers();
	SetUpdateFlags();
END_IF

CheckUpdateFlags();
IF (xInitRunning_Module_1 = FALSE) AND (xDataInUpdated = FALSE) THEN
	IF (mbxModule_1.bStatus.0) THEN
		SendValueRequest();
	END_IF
END_IF

IF (xInitRunning_Module_1 = FALSE) AND (mbxModule_1.bStatus.0) THEN
	xSetOnce := TRUE;
	xDataInUpdated := FALSE;
	IF ((NOT FuMemCompare(ADR(nvoStatusLast), ADR(nvoStatus), ADR(nvoStatus.bStatusInformation) - ADR(nvoStatus))) OR (nvoStatus.bStatusInformation.7 = TRUE) OR (nvoStatusLast.bInternalUseOnly.1 = TRUE)) THEN
		FuSnvtObjStatusToRaw(ADR(nvoStatus), ADR(OutDataTelegram_Module_1[2]));

		bNvAbsoluteIdx := bNvStartIndex + bObjectIndex + (1 * bLmoCount);

		IF (FuDoNvoUpdate_Module_1(ADR(nvoStatus), ADR(nvoStatusLast), ADR(nvoStatus.bInternalUseOnly), ADR(nvoStatusLast.bInternalUseOnly), ADR(nvoStatus.bStatusInformation), bNvAbsoluteIdx, 6, SIZEOF(nvoStatus)) = FALSE) THEN
			RETURN;
		END_IF
	END_IF
	IF ((NOT FuMemCompare(ADR(nvoFileStatLast), ADR(nvoFileStat), ADR(nvoFileStat.bStatusInformation) - ADR(nvoFileStat))) OR (nvoFileStat.bStatusInformation.7 = TRUE) OR (nvoFileStatLast.bInternalUseOnly.1 = TRUE)) THEN
		FuSnvtFileStatusToRaw(ADR(nvoFileStat), ADR(OutDataTelegram_Module_1[2]));

		bNvAbsoluteIdx := bNvStartIndex + bObjectIndex + (3 * bLmoCount);

		IF (FuDoNvoUpdate_Module_1(ADR(nvoFileStat), ADR(nvoFileStatLast), ADR(nvoFileStat.bInternalUseOnly), ADR(nvoFileStatLast.bInternalUseOnly), ADR(nvoFileStat.bStatusInformation), bNvAbsoluteIdx, 27, SIZEOF(nvoFileStat)) = FALSE) THEN
			RETURN;
		END_IF
	END_IF

END_IF
END_FUNCTION_BLOCK
ACTION CachePointers:
;
END_ACTION
ACTION CheckUpdateFlags:
xDataInUpdated := (NOT nviRequest.bInternalUseOnly.0) AND (NOT nviFileReq.bInternalUseOnly.0) AND (NOT nviFilePos.bInternalUseOnly.0) AND TRUE;
END_ACTION
ACTION DataReceived:
cmd := InDataTelegram_Module_1[0];
IF (cmd = M2C_NVI_UPDT_OCCD) OR (cmd = M2C_NV_VALUE_RSP) OR (cmd = M2C_NVI_UPDT_TOUT) THEN
	bNvRelativeIdx := (InDataTelegram_Module_1[1] - bNvStartIndex - bObjectIndex) / bLmoCount;
	CASE bNvRelativeIdx OF
	0:
		IF (cmd = M2C_NVI_UPDT_OCCD) OR (cmd = M2C_NV_VALUE_RSP) THEN
			IF (unLastLen_mbxModule_1 = (2 + 3)) THEN
				FuRawToSnvtObjRequest(ADR(InDataTelegram_Module_1[2]), ADR(nviRequest));
				nviRequest.bInternalUseOnly.0 := FALSE;
				nviRequest.bStatusInformation := FuInkrementNviStatus(nviRequest.bStatusInformation);
			ELSIF (unLastLen_mbxModule_1 = 2) THEN
				nviRequest.bStatusInformation := FuInkrementNviStatus(nviRequest.bStatusInformation);
			END_IF
		ELSIF (cmd = M2C_NVI_UPDT_TOUT) THEN
			IF (unLastLen_mbxModule_1 = 3) THEN
				nviRequest.bStatusInformation.4 := BYTE_TO_BOOL(InDataTelegram_Module_1[2]);
			END_IF
		END_IF
	2:
		IF (cmd = M2C_NVI_UPDT_OCCD) OR (cmd = M2C_NV_VALUE_RSP) THEN
			IF (unLastLen_mbxModule_1 = (2 + 12)) THEN
				FuRawToSnvtFileReq(ADR(InDataTelegram_Module_1[2]), ADR(nviFileReq));
				nviFileReq.bInternalUseOnly.0 := FALSE;
				nviFileReq.bStatusInformation := FuInkrementNviStatus(nviFileReq.bStatusInformation);
			ELSIF (unLastLen_mbxModule_1 = 2) THEN
				nviFileReq.bStatusInformation := FuInkrementNviStatus(nviFileReq.bStatusInformation);
			END_IF
		ELSIF (cmd = M2C_NVI_UPDT_TOUT) THEN
			IF (unLastLen_mbxModule_1 = 3) THEN
				nviFileReq.bStatusInformation.4 := BYTE_TO_BOOL(InDataTelegram_Module_1[2]);
			END_IF
		END_IF
	4:
		IF (cmd = M2C_NVI_UPDT_OCCD) OR (cmd = M2C_NV_VALUE_RSP) THEN
			IF (unLastLen_mbxModule_1 = (2 + 6)) THEN
				FuRawToSnvtFilePos(ADR(InDataTelegram_Module_1[2]), ADR(nviFilePos));
				nviFilePos.bInternalUseOnly.0 := FALSE;
				nviFilePos.bStatusInformation := FuInkrementNviStatus(nviFilePos.bStatusInformation);
			ELSIF (unLastLen_mbxModule_1 = 2) THEN
				nviFilePos.bStatusInformation := FuInkrementNviStatus(nviFilePos.bStatusInformation);
			END_IF
		ELSIF (cmd = M2C_NVI_UPDT_TOUT) THEN
			IF (unLastLen_mbxModule_1 = 3) THEN
				nviFilePos.bStatusInformation.4 := BYTE_TO_BOOL(InDataTelegram_Module_1[2]);
			END_IF
		END_IF

	END_CASE
ELSIF (cmd = M2C_CP_VALUE_RSP) THEN
	wCpRelativeIdx := ((InDataTelegram_Module_1[1] + InDataTelegram_Module_1[2] * 256) - wCpStartIndex - bObjectIndex) / bLmoCount;
	CASE wCpRelativeIdx OF

	END_CASE
END_IF
END_ACTION
ACTION ResetNviUpdate:
nviRequest.bStatusInformation := nviRequest.bStatusInformation AND 16#F8;
nviFileReq.bStatusInformation := nviFileReq.bStatusInformation AND 16#F8;
nviFilePos.bStatusInformation := nviFilePos.bStatusInformation AND 16#F8;
;
END_ACTION
ACTION SendValueRequest:
IF (FuSendNviValueReq_Module_1(ADR(nviRequest.bInternalUseOnly), bNvStartIndex + bObjectIndex + (0 * bLmoCount)) = FALSE) THEN
	RETURN;
END_IF

IF (FuSendNviValueReq_Module_1(ADR(nviFileReq.bInternalUseOnly), bNvStartIndex + bObjectIndex + (2 * bLmoCount)) = FALSE) THEN
	RETURN;
END_IF

IF (FuSendNviValueReq_Module_1(ADR(nviFilePos.bInternalUseOnly), bNvStartIndex + bObjectIndex + (4 * bLmoCount)) = FALSE) THEN
	RETURN;
END_IF

;
END_ACTION
ACTION SetUpdateFlags:
nviRequest.bInternaluseOnly.0 := TRUE;
nvoStatusLast.bInternaluseOnly.1 := TRUE;
nvoStatusLast.bInternaluseOnly.7 := FALSE;
nviFileReq.bInternaluseOnly.0 := TRUE;
nvoFileStatLast.bInternaluseOnly.1 := TRUE;
nvoFileStatLast.bInternaluseOnly.7 := FALSE;
nviFilePos.bInternaluseOnly.0 := TRUE;
;
END_ACTION

(* POU LON/Shared/Internal/FuSnvtObjStatusToRaw, ST *)
FUNCTION FuSnvtObjStatusToRaw : BOOL
(******************************************)
(* Automatic generated code, do not edit! *)
(******************************************)
VAR_INPUT
	NvDataIn :  POINTER TO typSnvtObjStatus;
	DataOut : POINTER TO ARRAY[0..5] OF BYTE;
END_VAR
VAR
END_VAR
DataOut^[0] := WORD_TO_BYTE(SHR(NvDataIn^.wObjectId, 8));
DataOut^[1] := WORD_TO_BYTE(NvDataIn^.wObjectId);

DataOut^[2] := NvDataIn^.bBitfieldByteOffset2;

DataOut^[3] := NvDataIn^.bBitfieldByteOffset3;

DataOut^[4] := NvDataIn^.bBitfieldByteOffset4;

DataOut^[5] := NvDataIn^.bBitfieldByteOffset5;

FuSnvtObjStatusToRaw := TRUE;
END_FUNCTION

(* POU LON/Module_1/Internal/FuDoNvoUpdate_Module_1, ST *)
FUNCTION FuDoNvoUpdate_Module_1 : BOOL
(******************************************)
(* Automatic generated code, do not edit! *)
(******************************************)
VAR_INPUT
	ptNvo : POINTER TO BYTE;
	ptNvoLast : POINTER TO BYTE;
	ptNvoInternalUse : POINTER TO BYTE;
	ptNvoLastInternalUse : POINTER TO BYTE;
	ptNvoStatusInformation : POINTER TO BYTE;
	bNvoIndex : BYTE;
	uiNvoLength : UINT;
	uiNvoVariableLength : UINT;
END_VAR
IF (ptNvoLastInternalUse^.1 = TRUE) AND (ptNvoStatusInformation^.7 = FALSE) THEN
	OutDataTelegram_Module_1[0] := C2M_NV_VALUE;
ELSE
	OutDataTelegram_Module_1[0] := C2M_NVO_PROPAGATE;
END_IF
OutDataTelegram_Module_1[1] := bNvoIndex;

mbxModule_1.bTxPrio := BOOL_TO_BYTE(ptNvoLastInternalUse^.7);
mbxModule_1.bTxProtID := 0;
mbxModule_1.pbTxData := ADR(OutDataTelegram_Module_1);
mbxModule_1.unTxLen := 2 + uiNvoLength;
mbxModule_1.MBX_SEND();

IF (mbxModule_1.nError <> MBX_OK) THEN
	FuDoNvoUpdate_Module_1 := FALSE;
	RETURN;
END_IF

ptNvoLastInternalUse^.1 := FALSE;
ptNvoInternalUse^ := ptNvoLastInternalUse^;
FuMemCopy(ptNvo, ptNvoLast, uiNvoVariableLength);

FuDoNvoUpdate_Module_1 := TRUE;
END_FUNCTION

(* POU LON/Shared/Internal/FuSnvtFileStatusToRaw, ST *)
FUNCTION FuSnvtFileStatusToRaw : BOOL
(******************************************)
(* Automatic generated code, do not edit! *)
(******************************************)
VAR_INPUT
	NvDataIn :  POINTER TO typSnvtFileStatus;
	DataOut : POINTER TO ARRAY[0..26] OF BYTE;
END_VAR
VAR
END_VAR
DataOut^[0] := NvDataIn^.bStatus;

DataOut^[1] := WORD_TO_BYTE(SHR(NvDataIn^.wNumberOfFiles, 8));
DataOut^[2] := WORD_TO_BYTE(NvDataIn^.wNumberOfFiles);

DataOut^[3] := WORD_TO_BYTE(SHR(NvDataIn^.wSelectedFile, 8));
DataOut^[4] := WORD_TO_BYTE(NvDataIn^.wSelectedFile);

DataOut^[5] := NvDataIn^.abAdr[0];
DataOut^[6] := NvDataIn^.abAdr[1];
DataOut^[7] := NvDataIn^.abAdr[2];
DataOut^[8] := NvDataIn^.abAdr[3];
DataOut^[9] := NvDataIn^.abAdr[4];
DataOut^[10] := NvDataIn^.abAdr[5];
DataOut^[11] := NvDataIn^.abAdr[6];
DataOut^[12] := NvDataIn^.abAdr[7];
DataOut^[13] := NvDataIn^.abAdr[8];
DataOut^[14] := NvDataIn^.abAdr[9];
DataOut^[15] := NvDataIn^.abAdr[10];
DataOut^[16] := NvDataIn^.abAdr[11];
DataOut^[17] := NvDataIn^.abAdr[12];
DataOut^[18] := NvDataIn^.abAdr[13];
DataOut^[19] := NvDataIn^.abAdr[14];
DataOut^[20] := NvDataIn^.abAdr[15];
DataOut^[21] := NvDataIn^.abAdr[16];
DataOut^[22] := NvDataIn^.abAdr[17];
DataOut^[23] := NvDataIn^.abAdr[18];
DataOut^[24] := NvDataIn^.abAdr[19];
DataOut^[25] := NvDataIn^.abAdr[20];
DataOut^[26] := NvDataIn^.abAdr[21];

FuSnvtFileStatusToRaw := TRUE;
END_FUNCTION

(* POU LON/Module_1/Internal/FuSendNviValueReq_Module_1, ST *)
FUNCTION FuSendNviValueReq_Module_1 : BOOL
(******************************************)
(* Automatic generated code, do not edit! *)
(******************************************)
VAR_INPUT
	ptInternalUseOnly : POINTER TO BYTE;
	bNvIndex : BYTE;
END_VAR
IF ptInternalUseOnly^.0 = TRUE THEN
	OutDataTelegram_Module_1[0] := C2M_NV_VALUE_QRY;
	OutDataTelegram_Module_1[1] := bNvIndex;

	mbxModule_1.bTxPrio := 1;
	mbxModule_1.bTxProtID := 0;
	mbxModule_1.pbTxData := ADR(OutDataTelegram_Module_1);
	mbxModule_1.unTxLen := 2;
	mbxModule_1.MBX_SEND();

	IF (mbxModule_1.nError <> MBX_OK) THEN
		FuSendNviValueReq_Module_1 := FALSE;
		RETURN;
	END_IF
	ptInternalUseOnly^.0 := FALSE;
END_IF

FuSendNviValueReq_Module_1 := TRUE;
END_FUNCTION

(* POU LON/Module_1/NV_Interface/Module_1_Virtualfunctionalblock, ST *)
FUNCTION_BLOCK Module_1_Virtualfunctionalblock
(******************************************)
(* Automatic generated code, do not edit! *)
(******************************************)
VAR_INPUT
	bObjectIndex : BYTE := 0;
	VT_Request : typSnvtObjRequest;
	VT_TimeSet : typSnvtTimeStamp;
	VT_AlarmSet : typSnvtAlarm;
	VT_HCC1_ModeSet : typSnvtHvacMode;
	VT_HCC1_TempSet : typSnvtTempP;
	VT_HCC1_SuppTemp : typSnvtTempP;
	VT_HCC2_ModeSet : typSnvtHvacMode;
	VT_HCC2_TempSet : typSnvtTempP;
	VT_HCC2_SuppTemp : typSnvtTempP;
	VT_HCC3_ModeSet : typSnvtHvacMode;
	VT_HCC3_TempSet : typSnvtTempP;
	VT_HCC3_SuppTemp : typSnvtTempP;
	VT_DHW_ModeSet : typSnvtHvacMode;
	VT_DHW_SetPoint : typSnvtTempP;
	VT_CFD_SetEnable : typSnvtSwitch;
	VT_CFD_SetMode : typSnvtHvacMode;
	VT_CFD_SetPoint : typSnvtTempP;
	VT_BOC_SetEnable : typSnvtSwitch;
	VT_BOC_SetMode : typSnvtHvacMode;
	VT_BOC_SetPoint : typSnvtTempP;

END_VAR
VAR_OUTPUT
	VT_Status : typSnvtObjStatus;
	VT_Alarm : typSnvtAlarm;
	VT_RlyState : typSnvtState;
	VT_HCC1_Mode : typSnvtHvacMode;
	VT_HCC1_Temp : typSnvtTempP;
	VT_HCC2_Mode : typSnvtHvacMode;
	VT_HCC2_Temp : typSnvtTempP;
	VT_HCC3_Mode : typSnvtHvacMode;
	VT_HCC3_Temp : typSnvtTempP;
	VT_DHW_ActTemp : typSnvtTempP;
	VT_DHW_TempSet : typSnvtTempP;
	VT_CFD_GetEnable : typSnvtSwitch;
	VT_CFD_Temp : typSnvtTempP;
	VT_CFD_SetTemp : typSnvtTempP;
	VT_BOC_GetEnable : typSnvtSwitch;
	VT_BOC_Temp : typSnvtTempP;
	VT_BOC_SetTemp : typSnvtTempP;

END_VAR
VAR
	xSetOnce : BOOL := TRUE;
	xDataInUpdated : BOOL := FALSE;
	VT_RequestLast: typSnvtObjRequest;
	VT_TimeSetLast: typSnvtTimeStamp;
	VT_AlarmSetLast: typSnvtAlarm;
	paNviSnvtHvacMode : ARRAY[0..2] OF POINTER TO typSnvtHvacMode;
	aNviSnvtHvacModeIndex : ARRAY[0..2] OF BYTE := 7,12,17;
	paNviSnvtTempP : ARRAY[0..8] OF POINTER TO typSnvtTempP;
	aNviSnvtTempPIndex : ARRAY[0..8] OF BYTE := 9,14,19,22,24,28,30,34,36;
	paNviSnvtSwitch : ARRAY[0..1] OF POINTER TO typSnvtSwitch;
	aNviSnvtSwitchIndex : ARRAY[0..1] OF BYTE := 26,32;
	paNvoSnvtHvacMode : ARRAY[0..5] OF POINTER TO typSnvtHvacMode;
	aNvoSnvtHvacModeIndex : ARRAY[0..5] OF BYTE := 6,11,16,21,27,33;
	aNvoSnvtHvacModeLast : ARRAY[0..5] OF typSnvtHvacMode;
	aNvoSnvtHvacModePriority : ARRAY[0..0] OF BYTE := 16#00;
	paNvoSnvtTempP : ARRAY[0..8] OF POINTER TO typSnvtTempP;
	aNvoSnvtTempPIndex : ARRAY[0..8] OF BYTE := 8,10,13,15,18,20,23,29,35;
	aNvoSnvtTempPLast : ARRAY[0..8] OF typSnvtTempP;
	aNvoSnvtTempPPriority : ARRAY[0..1] OF BYTE := 16#00, 16#00;
	paNvoSnvtSwitch : ARRAY[0..1] OF POINTER TO typSnvtSwitch;
	aNvoSnvtSwitchIndex : ARRAY[0..1] OF BYTE := 25,31;
	aNvoSnvtSwitchLast : ARRAY[0..1] OF typSnvtSwitch;
	aNvoSnvtSwitchPriority : ARRAY[0..0] OF BYTE := 16#00;

	cmd : BYTE;
	z : INT;
	bNvRelativeIdx : BYTE;
	bNvAbsoluteIdx : BYTE;
	wCpRelativeIdx : WORD;
	wCpAbsoluteIdx : WORD;
END_VAR
VAR CONSTANT
	bNvStartIndex : BYTE := 5;
	wCpStartIndex : WORD := 65535;
	bLmoCount : BYTE := 1;
END_VAR
IF (xInitRunning_Module_1 = TRUE) AND (xSetOnce = TRUE) THEN
	xSetOnce := FALSE;
	CachePointers();
	SetUpdateFlags();
END_IF

CheckUpdateFlags();
IF (xInitRunning_Module_1 = FALSE) AND (xDataInUpdated = FALSE) THEN
	IF (mbxModule_1.bStatus.0) THEN
		SendValueRequest();
	END_IF
END_IF

IF (xInitRunning_Module_1 = FALSE) AND (mbxModule_1.bStatus.0) THEN
	xSetOnce := TRUE;
	xDataInUpdated := FALSE;
	IF ((NOT FuMemCompare(ADR(VT_RequestLast), ADR(VT_Request), ADR(VT_Request.bStatusInformation) - ADR(VT_Request))) OR (VT_Request.bStatusInformation.7 = TRUE) OR (VT_RequestLast.bInternalUseOnly.1 = TRUE)) THEN
		FuSnvtObjRequestToRaw(ADR(VT_Request), ADR(OutDataTelegram_Module_1[2]));

		bNvAbsoluteIdx := bNvStartIndex + bObjectIndex + (0 * bLmoCount);

		IF (FuDoNvoUpdate_Module_1(ADR(VT_Request), ADR(VT_RequestLast), ADR(VT_Request.bInternalUseOnly), ADR(VT_RequestLast.bInternalUseOnly), ADR(VT_Request.bStatusInformation), bNvAbsoluteIdx, 3, SIZEOF(VT_Request)) = FALSE) THEN
			RETURN;
		END_IF
	END_IF
	IF ((NOT FuMemCompare(ADR(VT_TimeSetLast), ADR(VT_TimeSet), ADR(VT_TimeSet.bStatusInformation) - ADR(VT_TimeSet))) OR (VT_TimeSet.bStatusInformation.7 = TRUE) OR (VT_TimeSetLast.bInternalUseOnly.1 = TRUE)) THEN
		FuSnvtTimeStampToRaw(ADR(VT_TimeSet), ADR(OutDataTelegram_Module_1[2]));

		bNvAbsoluteIdx := bNvStartIndex + bObjectIndex + (2 * bLmoCount);

		IF (FuDoNvoUpdate_Module_1(ADR(VT_TimeSet), ADR(VT_TimeSetLast), ADR(VT_TimeSet.bInternalUseOnly), ADR(VT_TimeSetLast.bInternalUseOnly), ADR(VT_TimeSet.bStatusInformation), bNvAbsoluteIdx, 7, SIZEOF(VT_TimeSet)) = FALSE) THEN
			RETURN;
		END_IF
	END_IF
	IF ((NOT FuMemCompare(ADR(VT_AlarmSetLast), ADR(VT_AlarmSet), ADR(VT_AlarmSet.bStatusInformation) - ADR(VT_AlarmSet))) OR (VT_AlarmSet.bStatusInformation.7 = TRUE) OR (VT_AlarmSetLast.bInternalUseOnly.1 = TRUE)) THEN
		FuSnvtAlarmToRaw(ADR(VT_AlarmSet), ADR(OutDataTelegram_Module_1[2]));

		bNvAbsoluteIdx := bNvStartIndex + bObjectIndex + (4 * bLmoCount);

		IF (FuDoNvoUpdate_Module_1(ADR(VT_AlarmSet), ADR(VT_AlarmSetLast), ADR(VT_AlarmSet.bInternalUseOnly), ADR(VT_AlarmSetLast.bInternalUseOnly), ADR(VT_AlarmSet.bStatusInformation), bNvAbsoluteIdx, 29, SIZEOF(VT_AlarmSet)) = FALSE) THEN
			RETURN;
		END_IF
	END_IF
	FOR z := 0 TO 5 DO
		IF ((NOT FuMemCompare(ADR(aNvoSnvtHvacModeLast[z]), paNvoSnvtHvacMode[z], ADR(paNvoSnvtHvacMode[z]^.bStatusInformation) - paNvoSnvtHvacMode[z])) OR (paNvoSnvtHvacMode[z]^.bStatusInformation.7 = TRUE) OR (aNvoSnvtHvacModeLast[z].bInternalUseOnly.1 = TRUE)) THEN
			FuSnvtHvacModeToRaw(paNvoSnvtHvacMode[z], ADR(OutDataTelegram_Module_1[2]));

			bNvAbsoluteIdx := bNvStartIndex + bObjectIndex + (aNvoSnvtHvacModeIndex[z] * bLmoCount);

			IF (FuDoNvoUpdate_Module_1(paNvoSnvtHvacMode[z], ADR(aNvoSnvtHvacModeLast[z]), ADR(paNvoSnvtHvacMode[z]^.bInternalUseOnly), ADR(aNvoSnvtHvacModeLast[z].bInternalUseOnly), ADR(paNvoSnvtHvacMode[z]^.bStatusInformation), bNvAbsoluteIdx, 1, SIZEOF(aNvoSnvtHvacModeLast[z])) = FALSE) THEN
				RETURN;
			END_IF
		END_IF
	END_FOR
	FOR z := 0 TO 8 DO
		IF ((NOT FuMemCompare(ADR(aNvoSnvtTempPLast[z]), paNvoSnvtTempP[z], ADR(paNvoSnvtTempP[z]^.bStatusInformation) - paNvoSnvtTempP[z])) OR (paNvoSnvtTempP[z]^.bStatusInformation.7 = TRUE) OR (aNvoSnvtTempPLast[z].bInternalUseOnly.1 = TRUE)) THEN
			FuSnvtTempPToRaw(paNvoSnvtTempP[z], ADR(OutDataTelegram_Module_1[2]));

			bNvAbsoluteIdx := bNvStartIndex + bObjectIndex + (aNvoSnvtTempPIndex[z] * bLmoCount);

			IF (FuDoNvoUpdate_Module_1(paNvoSnvtTempP[z], ADR(aNvoSnvtTempPLast[z]), ADR(paNvoSnvtTempP[z]^.bInternalUseOnly), ADR(aNvoSnvtTempPLast[z].bInternalUseOnly), ADR(paNvoSnvtTempP[z]^.bStatusInformation), bNvAbsoluteIdx, 2, SIZEOF(aNvoSnvtTempPLast[z])) = FALSE) THEN
				RETURN;
			END_IF
		END_IF
	END_FOR
	FOR z := 0 TO 1 DO
		IF ((NOT FuMemCompare(ADR(aNvoSnvtSwitchLast[z]), paNvoSnvtSwitch[z], ADR(paNvoSnvtSwitch[z]^.bStatusInformation) - paNvoSnvtSwitch[z])) OR (paNvoSnvtSwitch[z]^.bStatusInformation.7 = TRUE) OR (aNvoSnvtSwitchLast[z].bInternalUseOnly.1 = TRUE)) THEN
			FuSnvtSwitchToRaw(paNvoSnvtSwitch[z], ADR(OutDataTelegram_Module_1[2]));

			bNvAbsoluteIdx := bNvStartIndex + bObjectIndex + (aNvoSnvtSwitchIndex[z] * bLmoCount);

			IF (FuDoNvoUpdate_Module_1(paNvoSnvtSwitch[z], ADR(aNvoSnvtSwitchLast[z]), ADR(paNvoSnvtSwitch[z]^.bInternalUseOnly), ADR(aNvoSnvtSwitchLast[z].bInternalUseOnly), ADR(paNvoSnvtSwitch[z]^.bStatusInformation), bNvAbsoluteIdx, 2, SIZEOF(aNvoSnvtSwitchLast[z])) = FALSE) THEN
				RETURN;
			END_IF
		END_IF
	END_FOR

